// NETWORK 3 (disabled)
//   b_goto_Az_done: ********************************Zero Velocity***************************************
// fb_start_goto_az1(CLK := b_goto_Az_done); // R_TRIG
// b_start_goto_az R= fb_start_goto_az1.Q;
// b_moving R= fb_start_goto_az1.Q;

// NETWORK 4 (disabled)
//   b_scc_goto: the command of goto a fixed position for all axises
// fb_blink_move_az(ENABLE := b_moving, TIMELOW := t#1000ms, TIMEHIGH := t#200ms); // BLINK
// b_scc_goto := fb_blink_move_az.OUT;

// NETWORK 5 (disabled)
//   b_remote_on: in the remote mode
//   b_local_on: in the local mode
//   b_scc_goto: the command of goto a fixed position for all axises
//   v_elevation: Virtual axis "v_elevation" with axis number 8
// fb_goto_El(
//     Execute := (b_remote_on OR b_local_on) AND b_scc_goto,
//     Position := r_goto_el,
//     Velocity := 650,
//     Acceleration := 20,
//     Deceleration := 20,
//     Axis := v_elevation,
//     Active => b_active_el); // MC_MoveAbsolute
// b_goto_El_done := fb_goto_El.Done;

// NETWORK 6
//   b_remote_on: in the remote mode
//   b_local_on: in the local mode
//   b_start_goto_az_tcp: the command of goto a fixed position for all axises
//   v_FeedIndexer: Virtual axis "v_polarization" with axis number 9
fb_goto_FI(
    Execute := (b_remote_on OR b_local_on) AND b_start_goto_az_tcp,
    Distance := r_goto_FI,
    Velocity := vel_move_FI,
    Acceleration := 0.017,
    Deceleration := 0.017,
    Axis := v_FeedIndexer,
    Active => b_active_FI); // MC_MoveRelative
b_goto_FI_done := fb_goto_FI.Done;

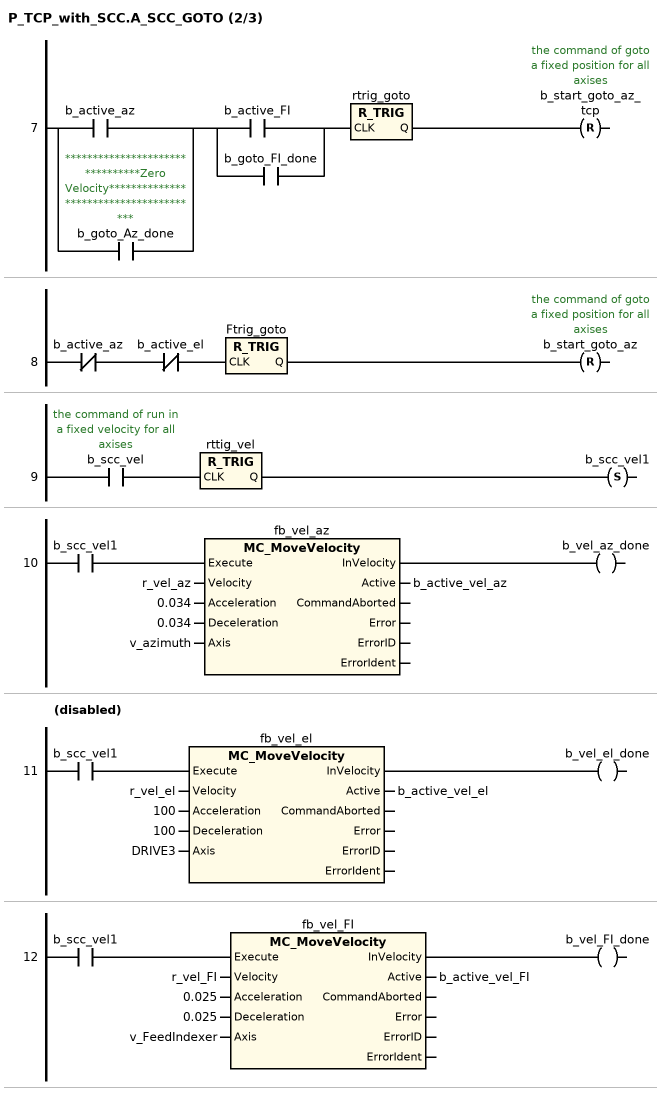
// NETWORK 7
//   b_goto_Az_done: ********************************Zero Velocity***************************************
//   b_start_goto_az_tcp: the command of goto a fixed position for all axises
rtrig_goto(CLK := (b_active_az OR b_goto_Az_done) AND (b_active_FI OR b_goto_FI_done)); // R_TRIG
b_start_goto_az_tcp R= rtrig_goto.Q;

// NETWORK 8
//   b_start_goto_az: the command of goto a fixed position for all axises
Ftrig_goto(CLK := NOT b_active_az AND NOT b_active_el); // R_TRIG
b_start_goto_az R= Ftrig_goto.Q;

// NETWORK 9
//   b_scc_vel: the command of run in a fixed velocity for all axises
rttig_vel(CLK := b_scc_vel); // R_TRIG
b_scc_vel1 S= rttig_vel.Q;

// NETWORK 10
//   r_vel_az: ************vel*************
//   v_azimuth: Virtual axis "v_azimuth" with axis number 7
fb_vel_az(
    Execute := b_scc_vel1,
    Velocity := r_vel_az,
    Acceleration := 0.034,
    Deceleration := 0.034,
    Axis := v_azimuth,
    Active => b_active_vel_az); // MC_MoveVelocity
b_vel_az_done := fb_vel_az.InVelocity;

// NETWORK 11 (disabled)
//   DRIVE3: Virtual axis "v_elevation" with axis number 8
// fb_vel_el(
//     Execute := b_scc_vel1,
//     Velocity := r_vel_el,
//     Acceleration := 100,
//     Deceleration := 100,
//     Axis := DRIVE3,
//     Active => b_active_vel_el); // MC_MoveVelocity
// b_vel_el_done := fb_vel_el.InVelocity;

// NETWORK 12
//   v_FeedIndexer: Virtual axis "v_polarization" with axis number 9
fb_vel_FI(
    Execute := b_scc_vel1,
    Velocity := r_vel_FI,
    Acceleration := 0.025,
    Deceleration := 0.025,
    Axis := v_FeedIndexer,
    Active => b_active_vel_FI); // MC_MoveVelocity
b_vel_FI_done := fb_vel_FI.InVelocity;

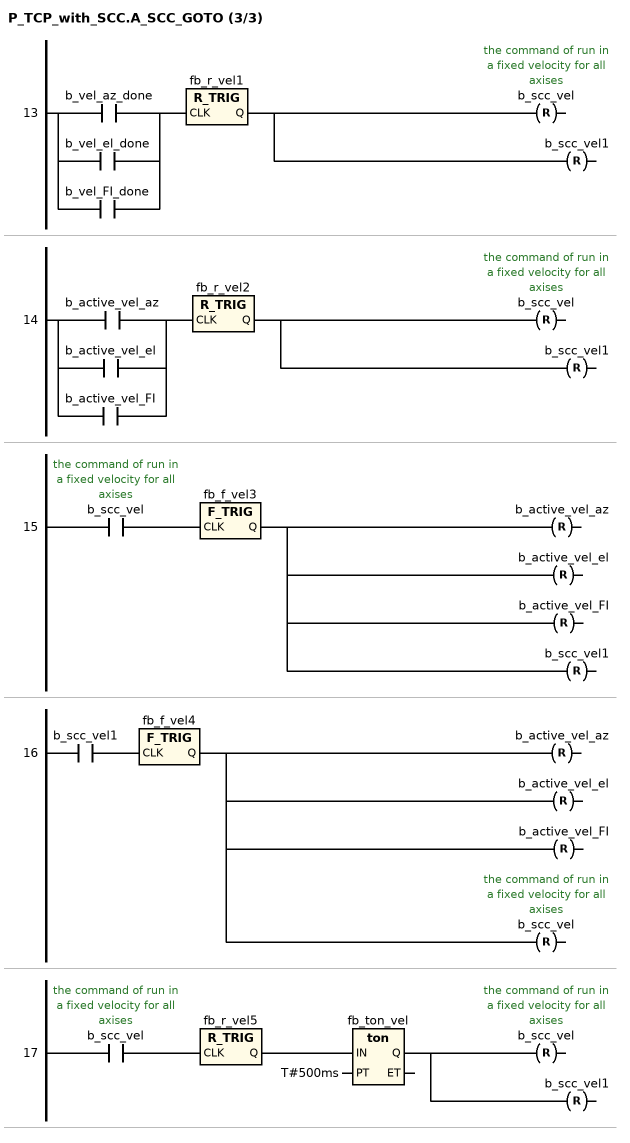
// NETWORK 13
//   b_scc_vel: the command of run in a fixed velocity for all axises
fb_r_vel1(CLK := b_vel_az_done OR b_vel_el_done OR b_vel_FI_done); // R_TRIG
b_scc_vel R= fb_r_vel1.Q;
b_scc_vel1 R= fb_r_vel1.Q;

// NETWORK 14
//   b_scc_vel: the command of run in a fixed velocity for all axises
fb_r_vel2(CLK := b_active_vel_az OR b_active_vel_el OR b_active_vel_FI); // R_TRIG
b_scc_vel R= fb_r_vel2.Q;
b_scc_vel1 R= fb_r_vel2.Q;

// NETWORK 15
//   b_scc_vel: the command of run in a fixed velocity for all axises
fb_f_vel3(CLK := b_scc_vel); // F_TRIG
b_active_vel_az R= fb_f_vel3.Q;
b_active_vel_el R= fb_f_vel3.Q;
b_active_vel_FI R= fb_f_vel3.Q;
b_scc_vel1 R= fb_f_vel3.Q;

// NETWORK 16
//   b_scc_vel: the command of run in a fixed velocity for all axises
fb_f_vel4(CLK := b_scc_vel1); // F_TRIG
b_active_vel_az R= fb_f_vel4.Q;
b_active_vel_el R= fb_f_vel4.Q;
b_active_vel_FI R= fb_f_vel4.Q;
b_scc_vel R= fb_f_vel4.Q;

// NETWORK 17
//   b_scc_vel: the command of run in a fixed velocity for all axises
fb_r_vel5(CLK := b_scc_vel); // R_TRIG
fb_ton_vel(IN := fb_r_vel5.Q, PT := T#500ms); // ton
b_scc_vel R= fb_ton_vel.Q;
b_scc_vel1 R= fb_ton_vel.Q;
END_ACTION

ACTION A_SCC_POWER:
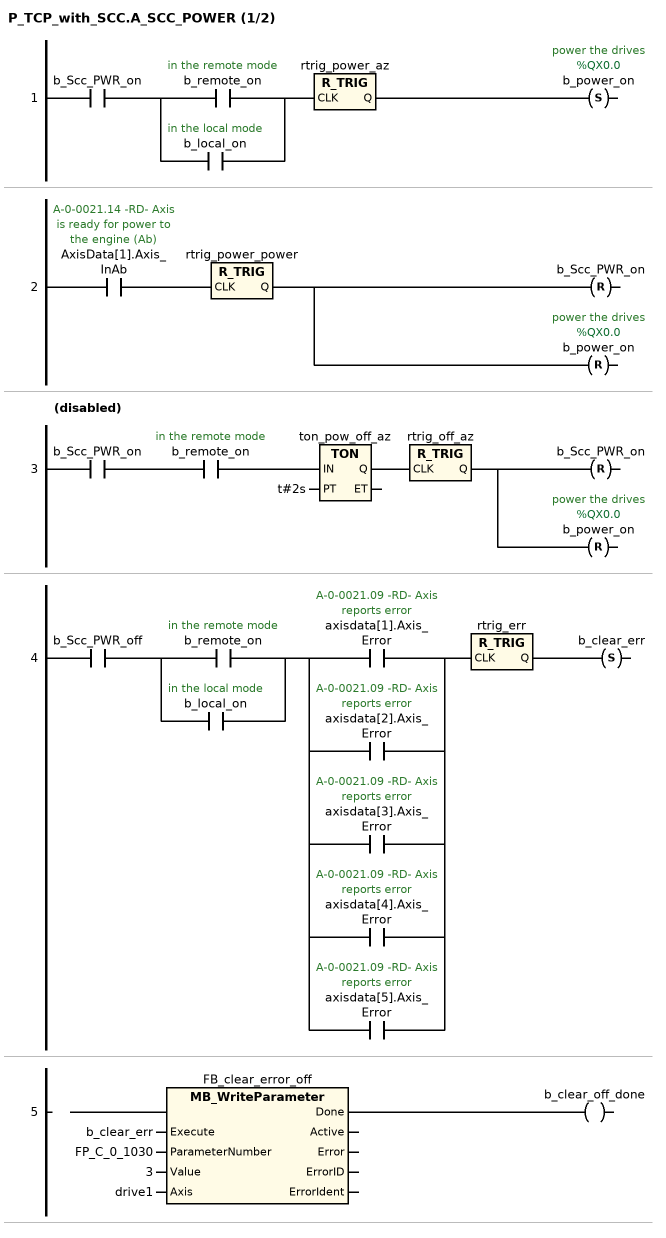
// NETWORK 1
//   b_remote_on: in the remote mode
//   b_local_on: in the local mode
//   b_power_on: power the drives | AT %QX0.0
rtrig_power_az(CLK := b_Scc_PWR_on AND (b_remote_on OR b_local_on)); // R_TRIG
b_power_on S= rtrig_power_az.Q;

// NETWORK 2
//   AxisData[1].Axis_InAb: A-0-0021.14 -RD- Axis is ready for power to the engine (Ab)
//   b_power_on: power the drives | AT %QX0.0
rtrig_power_power(CLK := AxisData[1].Axis_InAb); // R_TRIG
b_Scc_PWR_on R= rtrig_power_power.Q;
b_power_on R= rtrig_power_power.Q;

// NETWORK 3 (disabled)
//   ton_pow_off_az: <<<<<<<<<<<<<<<<<<<<<<<<<<<<<<<<<<<<<<<<<<<<<<<<<<<power>>>>>>>>>>>>>>>>>>>>>>>>>>>>>>>>>>>>
//   b_remote_on: in the remote mode
//   b_power_on: power the drives | AT %QX0.0
// ton_pow_off_az(IN := b_Scc_PWR_on AND b_remote_on, PT := t#2s); // TON
// rtrig_off_az(CLK := ton_pow_off_az.Q); // R_TRIG
// b_Scc_PWR_on R= rtrig_off_az.Q;
// b_power_on R= rtrig_off_az.Q;

// NETWORK 4
//   b_remote_on: in the remote mode
//   b_local_on: in the local mode
//   axisdata[1].Axis_Error: A-0-0021.09 -RD- Axis reports error
//   axisdata[2].Axis_Error: A-0-0021.09 -RD- Axis reports error
//   axisdata[3].Axis_Error: A-0-0021.09 -RD- Axis reports error
//   axisdata[4].Axis_Error: A-0-0021.09 -RD- Axis reports error
//   axisdata[5].Axis_Error: A-0-0021.09 -RD- Axis reports error
rtrig_err(CLK := b_Scc_PWR_off AND (b_remote_on OR b_local_on) AND (axisdata[1].Axis_Error OR axisdata[2].Axis_Error OR axisdata[3].Axis_Error OR axisdata[4].Axis_Error OR axisdata[5].Axis_Error)); // R_TRIG
b_clear_err S= rtrig_err.Q;

// NETWORK 5
//   FP_C_0_1030: Command: Clear all control errors
//   drive1: Real axis "Drive1" with axis number 1
FB_clear_error_off(Execute := b_clear_err, ParameterNumber := FP_C_0_1030, Value := 3, Axis := drive1); // MB_WriteParameter
b_clear_off_done := FB_clear_error_off.Done;

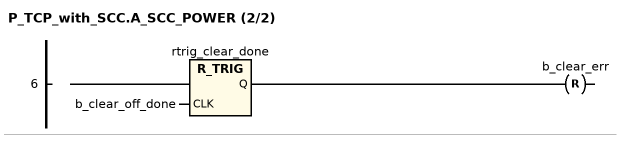
// NETWORK 6
rtrig_clear_done(CLK := b_clear_off_done); // R_TRIG
b_clear_err R= rtrig_clear_done.Q;
END_ACTION

ACTION A_SCC_STOP:
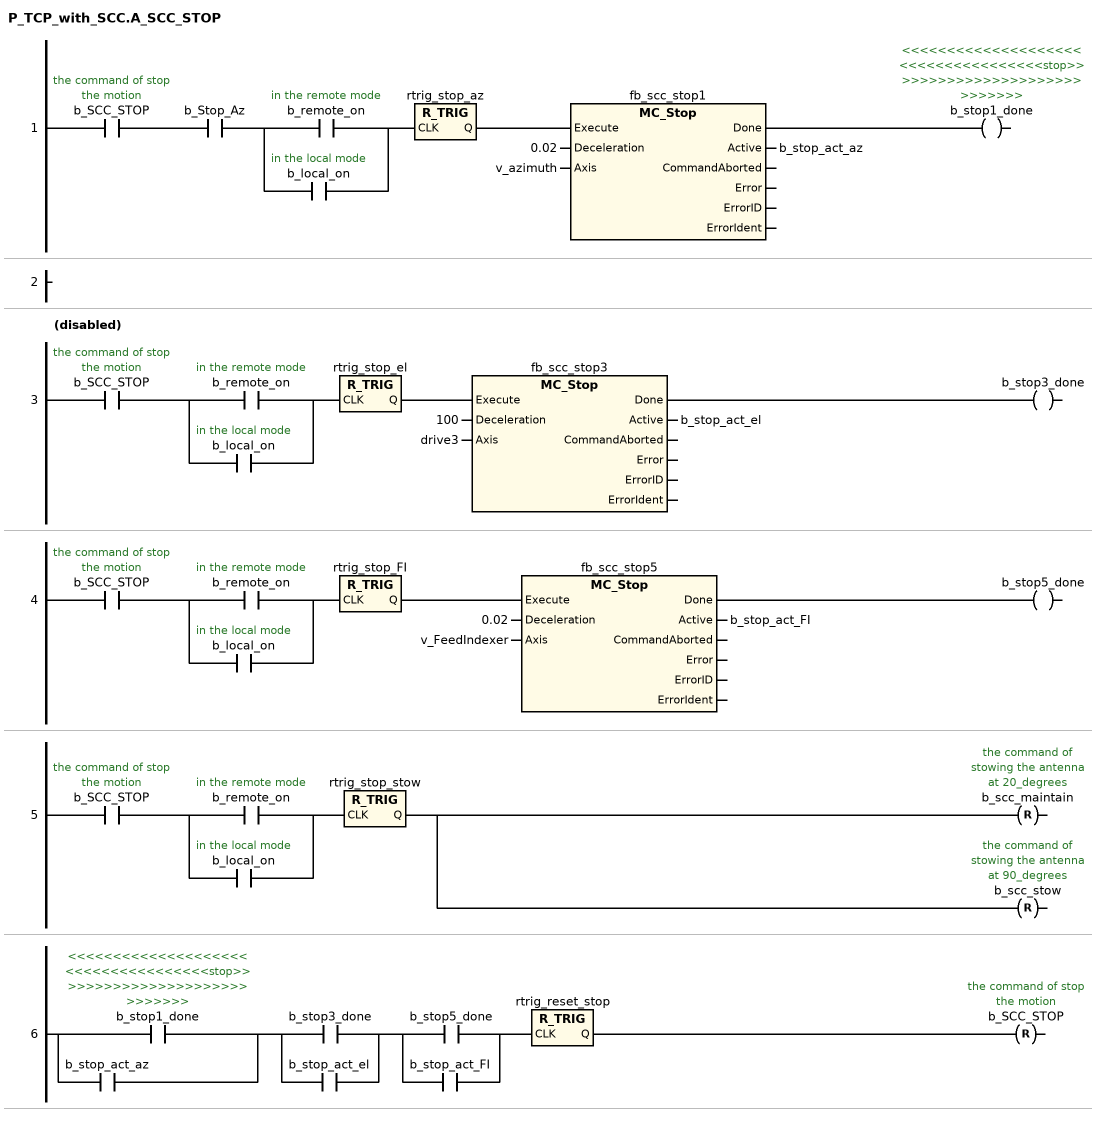
// NETWORK 1
//   b_SCC_STOP: the command of stop the motion
//   b_remote_on: in the remote mode
//   b_local_on: in the local mode
//   v_azimuth: Virtual axis "v_azimuth" with axis number 7
//   b_stop1_done: <<<<<<<<<<<<<<<<<<<<<<<<<<<<<<<<<<<<stop>>>>>>>>>>>>>>>>>>>>>>>>>>>>>
rtrig_stop_az(CLK := b_SCC_STOP AND b_Stop_Az AND (b_remote_on OR b_local_on)); // R_TRIG
fb_scc_stop1(Execute := rtrig_stop_az.Q, Deceleration := 0.02, Axis := v_azimuth, Active => b_stop_act_az); // MC_Stop
b_stop1_done := fb_scc_stop1.Done;

// NETWORK 2

// NETWORK 3 (disabled)
//   b_SCC_STOP: the command of stop the motion
//   b_remote_on: in the remote mode
//   b_local_on: in the local mode
//   drive3: Virtual axis "v_elevation" with axis number 8
// rtrig_stop_el(CLK := b_SCC_STOP AND (b_remote_on OR b_local_on)); // R_TRIG
// fb_scc_stop3(Execute := rtrig_stop_el.Q, Deceleration := 100, Axis := drive3, Active => b_stop_act_el); // MC_Stop
// b_stop3_done := fb_scc_stop3.Done;

// NETWORK 4
//   b_SCC_STOP: the command of stop the motion
//   b_remote_on: in the remote mode
//   b_local_on: in the local mode
//   v_FeedIndexer: Virtual axis "v_polarization" with axis number 9
rtrig_stop_FI(CLK := b_SCC_STOP AND (b_remote_on OR b_local_on)); // R_TRIG
fb_scc_stop5(
    Execute := rtrig_stop_FI.Q,
    Deceleration := 0.02,
    Axis := v_FeedIndexer,
    Active => b_stop_act_FI); // MC_Stop
b_stop5_done := fb_scc_stop5.Done;

// NETWORK 5
//   b_SCC_STOP: the command of stop the motion
//   b_remote_on: in the remote mode
//   b_local_on: in the local mode
//   b_scc_maintain: the command of stowing the antenna at 20_degrees
//   b_scc_stow: the command of stowing the antenna at 90_degrees
rtrig_stop_stow(CLK := b_SCC_STOP AND (b_remote_on OR b_local_on)); // R_TRIG
b_scc_maintain R= rtrig_stop_stow.Q;
b_scc_stow R= rtrig_stop_stow.Q;

// NETWORK 6
//   b_stop1_done: <<<<<<<<<<<<<<<<<<<<<<<<<<<<<<<<<<<<stop>>>>>>>>>>>>>>>>>>>>>>>>>>>>>
//   b_SCC_STOP: the command of stop the motion
rtrig_reset_stop(CLK := (b_stop1_done OR b_stop_act_az) AND (b_stop3_done OR b_stop_act_el) AND (b_stop5_done OR b_stop_act_FI)); // R_TRIG
b_SCC_STOP R= rtrig_reset_stop.Q;
END_ACTION

ACTION A_SEND:
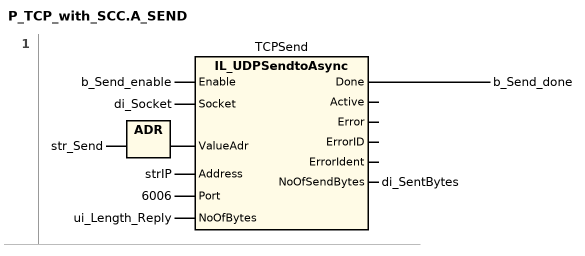
// NETWORK 1
TCPSend(
    Enable := b_Send_enable,
    Socket := di_Socket,
    ValueAdr := ADR(str_Send),
    Address := strIP,
    Port := 6006,
    NoOfBytes := ui_Length_Reply,
    NoOfSendBytes => di_SentBytes); // IL_UDPSendtoAsync
b_Send_done := TCPSend.Done;
END_ACTION

END_PROGRAM

// IndraMotionMlc1/Application/POUs/TCP/Message/FB_add_vector
(* the function block is programmed for adding points to trajectory stack.
The input variables is type of string,and the output vaiable is the reply for TCP*)
FUNCTION_BLOCK FB_add_vector
VAR_INPUT
	str_MJD:STRING;
	str_Azimuth:STRING;
	str_Elevation:STRING;
	str_FeedIndexer:STRING;
END_VAR
VAR_OUTPUT
	key:STRING;
END_VAR
VAR
(*(<<<<<<<<<<the transition variables>>>>>>>>>>>>>*)
	lreal_MJD: LREAL;
	real_azimuth: LREAL;
	real_elevation: LREAL;
	real_FeedIndexer: LREAL;
	tempAz:LREAL;
	tempEl:LREAL;
	temp_sin_Ao_C4:LREAL;
	temp_cos_Ao_C4:LREAL;
	temp_tanEo: LREAL;
	temp_sinE0:LREAL;
	temp_cosE0:LREAL;
	temp1:LREAL;
	temp2:LREAL;
	temp_R_sin_Ao_C4:LREAL;
	temp_R_cos_Ao_C4:LREAL;
	temp_R_tanEo:LREAL;
	temp_R_cosE0:LREAL;
	temp_R_sinE0:LREAL;
	temp1_exp:LREAL;
	temp2_exp:LREAL;
	new_Az:LREAL;
	new_El:LREAL;
	k:DINT;
	deltaAZ:LREAL:=0.0;
	deltaEL:LREAL:=0.0;
	aaaa:LREAL;
	bbbb:LREAL;
	test_1: LREAL;
END_VAR

(*lreal_MJD:=STRING_TO_LREAL(str_MJD)-0.000000076;*)(*set the ahead time for 6.6ms,so that the following error will be 0*)
// Assuming that for SKAO lreal_MJD will contain the TAIoffset. 
lreal_MJD:=STRING_TO_LREAL(str_MJD);(*after gunner change P41 into 100ms,so the aheed time must be added by 50ms.(56.5ms)*)

real_azimuth:=STRING_TO_LREAL(str_Azimuth);
real_Elevation:=STRING_TO_LREAL(str_Elevation);
real_FeedIndexer:=STRING_TO_REAL(str_FeedIndexer);
deltaAZ:=0.0;
deltaEL:=0.0;
	tempAz:=real_azimuth;
    tempEl:=real_Elevation;
(* This pointing model is not used for SKAO 
  		FOR k:=1 TO 3 BY 1 DO
        temp_sin_Ao_C4:=SIN(deg2rad(tempAz-C4));
        temp_cos_Ao_C4:=COS(deg2rad(tempAz-C4));
        temp_tanEo:=TAN(deg2rad(tempEl));
        temp_cosE0:=COS(deg2rad(tempEl));
        temp_sinE0:=SIN(deg2rad(tempEl));
        temp1:=tempAz-(C1+C3*temp_sin_Ao_C4*temp_tanEo+C5*temp_tanEo+C6/temp_cosE0);
        temp2:=tempEl-(C2+C3*temp_cos_Ao_C4+C7*temp_cosE0);
        temp_R_sin_Ao_C4:=SIN(deg2rad(temp1-C4));
        temp_R_cos_Ao_C4:=COS(deg2rad(temp1-C4));
        temp_R_tanEo:=TAN(deg2rad(temp2));
        temp_R_cosE0:=COS(deg2rad(temp2));
        temp_R_sinE0:=SIN(deg2rad(temp2));
        temp1_exp:=temp1+C1+C3*temp_R_sin_Ao_C4*temp_R_tanEo+C5*temp_R_tanEo+C6/temp_R_cosE0;
        temp2_exp:=temp2+C2+C3*temp_R_cos_Ao_C4+C7*temp_R_cosE0;
        deltaAz:=real_azimuth-temp1_exp;
        deltaEl:=real_Elevation-temp2_exp;
        tempAz:=tempAz+deltaAz;
        tempEl:=tempEl+deltaEl;
    END_FOR;
	*)
	new_Az:=temp1;
//	new_El:=Encoder_to_motor(temp2);
	new_El:=temp2;
	aaaa:=new_Az-real_azimuth;
	bbbb:=new_El-real_Elevation;
(*<<<<<<<<<<<<<<<<<<<<<<<<<<<<<<<judgement according to ICD document>>>>>>>>>>>>>>>>>>>>>>>>>>>>>>>*)

test_1:=lreal_MJD-lr_TAIoffset_current;
IF (lreal_MJD-lr_TAIoffset_current)>0.001 THEN	
IF real_azimuth>=-270 AND real_azimuth<=270 AND real_elevation>=15 AND real_elevation<=90 AND real_FeedIndexer>=0 AND real_FeedIndexer<=180 THEN
	IF lreal_MJD> (track_table[i_End].TAIoffset) THEN
		IF i_num_stack_left<i_total THEN
			IF track_table[i_end].TAIoffset<>0 THEN
				i_end:=F_I_number(i_end+1);
			END_IF;
			key:='OK';
			track_table[i_End].TAIoffset:=lreal_MJD;
			track_table[i_End].Azimuth:= new_Az;//-0.2884;
			track_table[i_End].Elevation:= real_Elevation;
			//track_table[i_End].FeedIndexer:= tempEl;
			//track_table[i_End].Elevation_ori:=temp2;
		ELSE
			key:='NAK - Stack is full';
		END_IF;
	ELSE
		key:='NAK - MJD is out of sequence';
	END_IF;
ELSE
	key:='NAK - One or more trkval coords are unreachable';
END_IF;
END_IF;

(*test_1:=lreal_MJD-lr_MJD_current;
IF (lreal_MJD-lr_MJD_current)>0.001 THEN	
IF real_azimuth>=-270 AND real_azimuth<=270 AND real_elevation>=15 AND real_elevation<=90 AND real_FeedIndexer>=0 AND real_FeedIndexer<=180 THEN
	IF lreal_MJD> (track_table[i_End].MJD) THEN
		IF i_num_stack_left<i_total THEN
			IF track_table[i_end].MJD<>0 THEN
				i_end:=F_I_number(i_end+1);
			END_IF;
			key:='OK';
			track_table[i_End].MJD:=lreal_MJD;
			track_table[i_End].Azimuth:= new_Az;//-0.2884;
			track_table[i_End].Elevation:= real_Elevation;
			track_table[i_End].FeedIndexer:= tempEl;
			track_table[i_End].Elevation_ori:=temp2;
		ELSE
			key:='NAK - Stack is full';
		END_IF;
	ELSE
		key:='NAK - MJD is out of sequence';
	END_IF;
ELSE
	key:='NAK - One or more trkval coords are unreachable';
END_IF;
END_IF; *)

END_FUNCTION_BLOCK

// IndraMotionMlc1/Application/AxisInterface/_Readme
PROGRAM _Readme
VAR
END_VAR

;
(*  English                              | Deutsch
Please do not change the programs and    | Bitte die Programme und Funktionsbausteine
function blocks in this folder. Updates  | in diesem Ordner nicht veraendern. Updates des
of the AxisInterface example project     | AxisInterface Besipielprojektes werden eine
will include an EXPORT-File with the     | EXPORT-Datei mit dem Inhalt dieses Ordners enthalten.
content of this folder.                  |
If you want to adapt the POUs, copy and  | Bei Anpassungen an den POEs bitte kopieren und 
rename it to avoid overwriting           | umbenennen, um ein Ueberschreiben zu vermeiden  *)

END_PROGRAM

// IndraMotionMlc1/Application/POUs/Useless/POU_1MS_Az_freq
PROGRAM POU_1MS_Az_freq
VAR
	r_cycle_count: INT;
	R_TRIG_count: R_TRIG;
	R_TRIG_count_1: R_TRIG;
	r_cycle_count_1: INT;
	MB_AxisDistanceAccumulator_1: MB_AxisDistanceAccumulator;
	bDisenable: BOOL;
	
	btestStart: BOOL;
	rdistance: REAL;
	
	CTU_1: CTU;
	bReset: BOOL;
	bSTOPPPP: BOOL;
	iTestint: REAL;
	rdistancediff: REAL;
	rdiffdistance: REAL;
	rOldDistance: REAL;
	bHometest: BOOL;
	MB_WriteRealParameter_1: MB_WriteRealParameter;
	rIniEncoderPos: REAL;

	R_TRIG_IniPos: R_TRIG;
	bStartRecord: BOOL;
	R_TRIG_condition: R_TRIG;
	teetet: BOOL;
	TON_1: TON;
	rAxis3ActVel: REAL;
	rSetAxis3Vel: REAL;
	
	R_TRIG_VEL: R_TRIG;
	test_motor_degree: LREAL;
	test_encoder: LREAL;
	
	postion_vel_array:ARRAY[1..201] OF LREAL;
	MJD_vel_array:ARRAY[1..201] OF LREAL;
	pos_vel_avg_array:ARRAY[1..181] OF LREAL;
	position_vel_i:INT:=0;
	position_vel_avg_i:INT:=0;
	position_vel_i_before:INT;
	r_temp1_pos:LREAL;
	r_temp1_mjd:LREAL;
	i_temp:INT;
	sum_vel:REAL;


	i_avg_1:INT:=0;
	i_avg_2:INT:=0;
	i_avg_3:INT:=0;
	temp_vel_avg_array:ARRAY[1..21] OF LREAL;
	sum_temp_vel:REAL;
	test1_temp:REAL;
	r_new_cmd_pos:REAL;
	r_new_cmd_pos_motor:REAL;
	r_new_cmd_pos_motor_relative:REAL;
	R_TRIG_pos_done:R_TRIG;
	R_TRIG_pos_done_2:R_TRIG;
	R_TRIG_pos_done_3:R_TRIG;
	R_TRIG_pos_done_4:R_TRIG;
	R_TRIG_pos_done_5:R_TRIG;
	R_TRIG_pos_done_6:R_TRIG;
	R_TRIG_pos_done_7:R_TRIG;
	R_TRIG_pos_done_8:R_TRIG;
	R_TRIG_pos_done_9:R_TRIG;
	R_TRIG_pos_done_10:R_TRIG;
	ton_pos2:TON;
	
	i_closeloop_max:INT:=10;
	i_time:INT:=0;
	r_difference:REAL;
	test_POWER_EL: BOOL;
	vel_blink:Util.BLINK;
	rSPEED1: REAL;
	ton_start_adjust_vel:TON;
	r_trig_start_adjust_vel: R_TRIG;
	r_vel_el_1:REAL;
	
	vel_freq:REAL;
	T_period:REAL:=2;
	temp_t:REAL:=0.0;
	start_to_freq:BOOL;
	temp_i:INT:=0;
	
	b_test_freq_resp: BOOL;
	b_in_normal_mode: BOOL := TRUE;
	b_test_pos_freq: BOOL;
	
	Frequency_vel:REAL:=0.5;
	test_vel_az1: REAL;
	A_sin:REAL;
END_VAR



	position_vel_i:= position_vel_i+1;
	IF position_vel_i>200 THEN
		position_vel_i:=1;
	END_IF
	postion_vel_array[position_vel_i]:=r_pos_el;
	MJD_vel_array[position_vel_i]:=lr_MJD_current;
	
	position_vel_i_before:=position_vel_i-100;
	IF position_vel_i_before<0 THEN
		position_vel_i_before:=position_vel_i_before+200;
	END_IF
	IF position_vel_i_before=0 THEN
		position_vel_i_before:=200;
	END_IF
		
	r_temp1_pos:=postion_vel_array[position_vel_i]-postion_vel_array[position_vel_i_before];
	r_temp1_mjd:=(MJD_vel_array[position_vel_i]-MJD_vel_array[position_vel_i_before])*86400;
	IF r_temp1_mjd= 0 THEN
		r_temp1_mjd :=1;
	END_IF
	position_vel_avg_i:=position_vel_avg_i+1;
	pos_vel_avg_array[position_vel_avg_i]:=r_temp1_pos/r_temp1_mjd;
	
	IF position_vel_avg_i = 180 THEN
		position_vel_avg_i:=0;
	END_IF
	
		sum_vel:=0;
	FOR i_temp :=1 TO 180 BY 1 DO
		sum_vel:=sum_vel+pos_vel_avg_array[i_temp];
	END_FOR
		r_vel_EL_temp:=sum_vel/180;
		
	i_avg_1:=i_avg_1+1;
	
	IF i_avg_1 =200 THEN
		i_avg_1:=0;
		i_avg_2:=i_avg_2+1;
		temp_vel_avg_array[i_avg_2]:=r_vel_EL_temp;
		IF i_avg_2>20 THEN
			i_avg_2:=0;
		END_IF		
	END_IF
	
		sum_temp_vel:=0;
	FOR i_avg_3 :=1 TO 20 BY 1 DO
		sum_temp_vel:=sum_temp_vel+temp_vel_avg_array[i_avg_3];
	END_FOR
		r_vel_EL:=sum_temp_vel/20;
	

		
	
	
//	r_vel_EL:=r_temp1_pos/r_temp1_mjd;
//	r_vel_EL:=(postion_vel_array[position_vel_i]-postion_vel_array[position_vel_i_before])/(MJD_vel_array[position_vel_i]-MJD_vel_array[position_vel_i_before])/86400;
	
	
	
	test_motor_degree:=Encoder_to_motor(test_encoder);
 
	//俯仰电机实时位置	
	r_pos_motor3:=axisdata[3].rActualPosition_i;	
	
	//俯仰电机位置累计
    rPosdiff:=RIL_Utilities.IL_GetModuloType04((axisdata[3].rActualPosition_i-roldposition),210000);
	//rPosdiff:=r_pos_motor3-roldposition;
	roldposition:=r_pos_motor3;
	r_length:=r_length+rPosdiff;
	
	CTU_1(CU:=axisdata[3].rActualPosition_i>180 , RESET:= bReset, PV:=10000 , Q=> , CV=> );
	CTU_1.CV;
	//测量Delta杆长值
	r_length_count := r_length/360/16.8*25;	
	
	//理论杆长
	Inir_Length:=SQRT(2984.1*2984.1+3150.6*3150.6-2*2984.1*3150.6*COS(r_pos_el*3.1415926/180));
	
	MB_AxisDistanceAccumulator_1(
	Enable:= bDisenable, 
	TotalDistance:= 1000000, 
	InOperation=> , 
	Error=> , 
	ErrorID=> , 
	ErrorIdent=> , 
	DistanceReached=> , 
	AccumulatedDistance=> r_length_Distance, 
	Axis:= Drive3);
/////////////**********上电设置编码器位置************////////////	
	R_TRIG_condition(CLK:=NOT TechBase.ImcStatus.Diag.Error 
							AND NOT arAxisStatus_gb[3].Admin.MODE_AH 
								AND ML_Base.AxisData[3].Axis_Inbb
									AND NOT bStartRecord, Q=> );
	IF  R_TRIG_condition.Q OR teetet  THEN 
		bHometest:=TRUE;
	END_IF
		MB_WriteRealParameter_1(
		Execute:= bHometest, 
		Done=> , 
		Active=> , 
		Error=> , 
		ErrorID=> , 
		ErrorIdent=> , 
		ParameterNumber:= ML_Base.FP_S_0_0052, 
		Value:= r_pos_motor3_Ini, 
		Axis:=Drive3 );	
	arAxisCtrl_gb[3].Admin.SetAbsRef:=MB_WriteRealParameter_1.Done;
		TON_1(IN:= MB_WriteRealParameter_1.Done, PT:=T#3S , Q=> , ET=> );
	//	R_TRIG_IniPos(CLK:= TON_1.Q, Q=> );
		IF TON_1.Q THEN 
			bStartRecord:=TRUE;
			bHometest:=FALSE;
		END_IF
		IF bStartRecord THEN
			r_pos_motor3_Ini:=axisdata[3].rActualPosition_i;
		END_IF
/////////////////**************************//////////////////////////	
 (*SIN_Curve  	
   iTestint:=iTestint+0.05;
   rdistance:=3600*SIN(iTestint*3.1415926/180);
   rdiffdistance:=rdistance-rOldDistance;
   rOldDistance:=rdistance;
   *) 
   
R_TRIG_VEL(CLK:=P_TCP_with_SCC.b_scc_vel1 , Q=> );	
IF R_TRIG_VEL.Q THEN 
	b_scc_vel1_temp:=TRUE;
END_IF

R_TRIG_pos_done(CLK:=arAxisStatus_gb[Drive3.AxisNo].Admin.CmdDone , Q=> );	
IF R_TRIG_pos_done.Q THEN 
	b_first_pos_done:=TRUE;
END_IF

R_TRIG_pos_done_2(CLK:=(arAxisStatus_gb[Drive3.AxisNo].Admin.CmdDone AND i_adjust_count=1) , Q=> );	
IF R_TRIG_pos_done_2.Q THEN 
	b_second_pos_done:=TRUE;
END_IF

R_TRIG_pos_done_3(CLK:=(arAxisStatus_gb[Drive3.AxisNo].Admin.CmdDone AND i_adjust_count=2) , Q=> );	
IF R_TRIG_pos_done_3.Q THEN 
	b_3rd_pos_done:=TRUE;
END_IF

R_TRIG_pos_done_4(CLK:=(arAxisStatus_gb[Drive3.AxisNo].Admin.CmdDone AND i_adjust_count=3) , Q=> );	
IF R_TRIG_pos_done_4.Q THEN 
	b_4th_pos_done:=TRUE;
END_IF

R_TRIG_pos_done_5(CLK:=(arAxisStatus_gb[Drive3.AxisNo].Admin.CmdDone AND i_adjust_count=4) , Q=> );	
IF R_TRIG_pos_done_5.Q THEN 
	b_5th_pos_done:=TRUE;
END_IF

R_TRIG_pos_done_6(CLK:=(arAxisStatus_gb[Drive3.AxisNo].Admin.CmdDone AND i_adjust_count=5) , Q=> );	
IF R_TRIG_pos_done_6.Q THEN 
	b_6th_pos_done:=TRUE;
END_IF

R_TRIG_pos_done_7(CLK:=(arAxisStatus_gb[Drive3.AxisNo].Admin.CmdDone AND i_adjust_count=6) , Q=> );	
IF R_TRIG_pos_done_7.Q THEN 
	b_7th_pos_done:=TRUE;
END_IF

R_TRIG_pos_done_8(CLK:=(arAxisStatus_gb[Drive3.AxisNo].Admin.CmdDone AND i_adjust_count=7) , Q=> );	
IF R_TRIG_pos_done_8.Q THEN 
	b_8th_pos_done:=TRUE;
END_IF

R_TRIG_pos_done_9(CLK:=(arAxisStatus_gb[Drive3.AxisNo].Admin.CmdDone AND i_adjust_count=8) , Q=> );	
IF R_TRIG_pos_done_9.Q THEN 
	b_9th_pos_done:=TRUE;
END_IF

R_TRIG_pos_done_10(CLK:=(arAxisStatus_gb[Drive3.AxisNo].Admin.CmdDone AND i_adjust_count=9) , Q=> );	
IF R_TRIG_pos_done_10.Q THEN 
	b_10th_pos_done:=TRUE;
END_IF

ton_pos2(IN:=b_second_pos_done,PT:=T#10S);
IF ton_pos2.Q THEN
adjust_delay:=TRUE;
END_IF

i_time:=i_time+1;
IF i_time>100 THEN
	i_time:=0;
END_IF

//IF i_time = 50 THEN
	IF TRUE THEN
	r_difference:=ABS(r_goto_el_I-r_pos_el);

IF b_in_positionMode  AND b_first_pos_done AND i_adjust_count=0 AND r_difference>0.0005 THEN

	r_new_cmd_pos:=2*r_goto_el_I-r_pos_el;
	r_new_cmd_pos_motor:=Encoder_to_motor(r_new_cmd_pos);
	r_new_cmd_pos_motor_relative:=Encoder_to_motor(r_goto_el_I)-Encoder_to_motor(ML_Base.AxisData[11].rActualPosition_i);
	r_goto_el_abs:=r_new_cmd_pos_motor;
	r_goto_el:=r_new_cmd_pos_motor_relative;
	b_in_positionMode:=FALSE;
	b_first_pos_done:=FALSE;
	b_second_pos_done:=FALSE;
	b_3rd_pos_done:=FALSE;
	b_4th_pos_done:=FALSE;
	b_5th_pos_done:=FALSE;
	b_6th_pos_done:=FALSE;
	b_7th_pos_done:=FALSE;
	b_8th_pos_done:=FALSE;
	b_9th_pos_done:=FALSE;
	b_10th_pos_done:=FALSE;
	i_adjust_count:=1;	
END_IF

IF i_adjust_count=1  AND b_second_pos_done AND  r_difference>0.0005 THEN

	r_new_cmd_pos:=2*r_goto_el_I-r_pos_el;
	r_new_cmd_pos_motor:=Encoder_to_motor(r_new_cmd_pos);
	r_new_cmd_pos_motor_relative:=Encoder_to_motor(r_goto_el_I)-Encoder_to_motor(ML_Base.AxisData[11].rActualPosition_i);
	r_goto_el_abs:=r_new_cmd_pos_motor;
	r_goto_el:=r_new_cmd_pos_motor_relative;
	b_in_positionMode:=FALSE;
	b_first_pos_done:=FALSE;
	b_second_pos_done:=FALSE;
	b_3rd_pos_done:=FALSE;
	b_4th_pos_done:=FALSE;
	b_5th_pos_done:=FALSE;
	b_6th_pos_done:=FALSE;
	b_7th_pos_done:=FALSE;
	b_8th_pos_done:=FALSE;
	b_9th_pos_done:=FALSE;
	b_10th_pos_done:=FALSE;
	adjust_delay:=FALSE;
	i_adjust_count:=2;
END_IF

IF i_adjust_count=2  AND b_3rd_pos_done AND r_difference>0.0005  THEN

	r_new_cmd_pos:=2*r_goto_el_I-r_pos_el;
	r_new_cmd_pos_motor:=Encoder_to_motor(r_new_cmd_pos);
	r_new_cmd_pos_motor_relative:=Encoder_to_motor(r_goto_el_I)-Encoder_to_motor(ML_Base.AxisData[11].rActualPosition_i);
	r_goto_el_abs:=r_new_cmd_pos_motor;
	r_goto_el:=r_new_cmd_pos_motor_relative;
	b_in_positionMode:=FALSE;
	b_first_pos_done:=FALSE;
	b_second_pos_done:=FALSE;
	b_3rd_pos_done:=FALSE;
	b_4th_pos_done:=FALSE;
	b_5th_pos_done:=FALSE;
	b_6th_pos_done:=FALSE;
	b_7th_pos_done:=FALSE;
	b_8th_pos_done:=FALSE;
	b_9th_pos_done:=FALSE;
	b_10th_pos_done:=FALSE;
	adjust_delay:=FALSE;
	i_adjust_count:=3;
END_IF

IF i_adjust_count=3  AND b_4th_pos_done AND r_difference>0.0005  THEN

	r_new_cmd_pos:=2*r_goto_el_I-r_pos_el;
	r_new_cmd_pos_motor:=Encoder_to_motor(r_new_cmd_pos);
	r_new_cmd_pos_motor_relative:=Encoder_to_motor(r_goto_el_I)-Encoder_to_motor(ML_Base.AxisData[11].rActualPosition_i);
	r_goto_el_abs:=r_new_cmd_pos_motor;
	r_goto_el:=r_new_cmd_pos_motor_relative;
	b_in_positionMode:=FALSE;
	b_first_pos_done:=FALSE;
	b_second_pos_done:=FALSE;
	b_3rd_pos_done:=FALSE;
	b_4th_pos_done:=FALSE;
	b_5th_pos_done:=FALSE;
	b_6th_pos_done:=FALSE;
	b_7th_pos_done:=FALSE;
	b_8th_pos_done:=FALSE;
	b_9th_pos_done:=FALSE;
	b_10th_pos_done:=FALSE;
	adjust_delay:=FALSE;
	i_adjust_count:=4;
END_IF

IF i_adjust_count=4  AND b_5th_pos_done AND r_difference>0.0005  THEN

	r_new_cmd_pos:=2*r_goto_el_I-r_pos_el;
	r_new_cmd_pos_motor:=Encoder_to_motor(r_new_cmd_pos);
	r_new_cmd_pos_motor_relative:=Encoder_to_motor(r_goto_el_I)-Encoder_to_motor(ML_Base.AxisData[11].rActualPosition_i);
	r_goto_el_abs:=r_new_cmd_pos_motor;
	r_goto_el:=r_new_cmd_pos_motor_relative;
	b_in_positionMode:=FALSE;
	b_first_pos_done:=FALSE;
	b_second_pos_done:=FALSE;
	b_3rd_pos_done:=FALSE;
	b_4th_pos_done:=FALSE;
	b_5th_pos_done:=FALSE;
	b_6th_pos_done:=FALSE;
	b_7th_pos_done:=FALSE;
	b_8th_pos_done:=FALSE;
	b_9th_pos_done:=FALSE;
	b_10th_pos_done:=FALSE;
	adjust_delay:=FALSE;
	i_adjust_count:=5;
END_IF
END_IF
(*
IF i_adjust_count=5  AND b_6th_pos_done THEN
	r_new_cmd_pos:=2*r_goto_el_I-r_pos_el;
	r_new_cmd_pos_motor:=Encoder_to_motor(r_new_cmd_pos);
	r_goto_el_abs:=r_new_cmd_pos_motor;
	b_in_positionMode:=FALSE;
	b_first_pos_done:=FALSE;
	b_second_pos_done:=FALSE;
	b_3rd_pos_done:=FALSE;
	b_4th_pos_done:=FALSE;
	b_5th_pos_done:=FALSE;
	b_6th_pos_done:=FALSE;
	b_7th_pos_done:=FALSE;
	b_8th_pos_done:=FALSE;
	b_9th_pos_done:=FALSE;
	b_10th_pos_done:=FALSE;
	adjust_delay:=FALSE;
	i_adjust_count:=6;
END_IF

IF i_adjust_count=6  AND b_7th_pos_done THEN
	r_new_cmd_pos:=2*r_goto_el_I-r_pos_el;
	r_new_cmd_pos_motor:=Encoder_to_motor(r_new_cmd_pos);
	r_goto_el_abs:=r_new_cmd_pos_motor;
	b_in_positionMode:=FALSE;
	b_first_pos_done:=FALSE;
	b_second_pos_done:=FALSE;
	b_3rd_pos_done:=FALSE;
	b_4th_pos_done:=FALSE;
	b_5th_pos_done:=FALSE;
	b_6th_pos_done:=FALSE;
	b_7th_pos_done:=FALSE;
	b_8th_pos_done:=FALSE;
	b_9th_pos_done:=FALSE;
	b_10th_pos_done:=FALSE;
	adjust_delay:=FALSE;
	i_adjust_count:=7;
END_IF

IF i_adjust_count=7  AND b_8th_pos_done THEN
	r_new_cmd_pos:=2*r_goto_el_I-r_pos_el;
	r_new_cmd_pos_motor:=Encoder_to_motor(r_new_cmd_pos);
	r_goto_el_abs:=r_new_cmd_pos_motor;
	b_in_positionMode:=FALSE;
	b_first_pos_done:=FALSE;
	b_second_pos_done:=FALSE;
	b_3rd_pos_done:=FALSE;
	b_4th_pos_done:=FALSE;
	b_5th_pos_done:=FALSE;
	b_6th_pos_done:=FALSE;
	b_7th_pos_done:=FALSE;
	b_8th_pos_done:=FALSE;
	b_9th_pos_done:=FALSE;
	b_10th_pos_done:=FALSE;
	adjust_delay:=FALSE;
	i_adjust_count:=8;
END_IF

IF i_adjust_count=8  AND b_9th_pos_done THEN
	r_new_cmd_pos:=2*r_goto_el_I-r_pos_el;
	r_new_cmd_pos_motor:=Encoder_to_motor(r_new_cmd_pos);
	r_goto_el_abs:=r_new_cmd_pos_motor;
	b_in_positionMode:=FALSE;
	b_first_pos_done:=FALSE;
	b_second_pos_done:=FALSE;
	b_3rd_pos_done:=FALSE;
	b_4th_pos_done:=FALSE;
	b_5th_pos_done:=FALSE;
	b_6th_pos_done:=FALSE;
	b_7th_pos_done:=FALSE;
	b_8th_pos_done:=FALSE;
	b_9th_pos_done:=FALSE;
	b_10th_pos_done:=FALSE;
	adjust_delay:=FALSE;
	i_adjust_count:=9;
END_IF

IF i_adjust_count=9  AND b_10th_pos_done THEN
	r_new_cmd_pos:=2*r_goto_el_I-r_pos_el;
	r_new_cmd_pos_motor:=Encoder_to_motor(r_new_cmd_pos);
	r_goto_el_abs:=r_new_cmd_pos_motor;
	b_in_positionMode:=FALSE;
	b_first_pos_done:=FALSE;
	b_second_pos_done:=FALSE;
	b_3rd_pos_done:=FALSE;
	b_4th_pos_done:=FALSE;
	b_5th_pos_done:=FALSE;
	b_6th_pos_done:=FALSE;
	b_7th_pos_done:=FALSE;
	b_8th_pos_done:=FALSE;
	b_9th_pos_done:=FALSE;
	b_10th_pos_done:=FALSE;
	adjust_delay:=FALSE;
	i_adjust_count:=10;
END_IF
*)
(*	
IF  arAxisStatus_gb[Drive3.AxisNo].Admin.CmdDone AND i_closeloop_count<i_closeloop_max THEN
	r_new_cmd_pos:=2*r_goto_el_I-r_pos_el;
	r_new_cmd_pos_motor:=Encoder_to_motor(r_new_cmd_pos);
	r_goto_el_abs:=r_new_cmd_pos_motor;
	arAxisStatus_gb[Drive3.AxisNo].Admin.CmdDone:=FALSE;
	i_closeloop_count:= i_closeloop_count+1;
END_IF
	IF i_closeloop_count>i_closeloop_max THEN
		i_closeloop_count:=i_closeloop_max;
	END_IF
*)
r_trig_start_adjust_vel(CLK:= b_scc_vel); 
IF r_trig_start_adjust_vel.Q THEN
	b_start_adjust_vel_temp:=TRUE;
END_IF

ton_start_adjust_vel(IN:=b_start_adjust_vel_temp,PT:=T#10S);
IF ton_start_adjust_vel.Q THEN
	b_start_adjust_vel_temp:=FALSE;
	b_start_adjust_vel:=TRUE;
END_IF

//	r_vel_el_1:= 0.00008*ML_Base.AxisData[11].rActualPosition_i*ML_Base.AxisData[11].rActualPosition_i - 0.0141*ML_Base.AxisData[11].rActualPosition_i + 1.6168;
//r_vel_el_1 := 0.0000000002*r_pos_el_v*r_pos_el_v*r_pos_el_v*r_pos_el_v*r_pos_el_v - 0.00000003*r_pos_el_v*r_pos_el_v*r_pos_el_v*r_pos_el_v + 0.000002*r_pos_el_v*r_pos_el_v*r_pos_el_v + 0.0001*r_pos_el_v*r_pos_el_v - 0.0187*r_pos_el_v + 1.6902;
r_vel_el_1 := 0.00000000928*r_pos_el_v*r_pos_el_v*r_pos_el_v*r_pos_el_v - 0.000002553*r_pos_el_v*r_pos_el_v*r_pos_el_v + 0.0003141*r_pos_el_v*r_pos_el_v - 0.02293*r_pos_el_v + 1.7235;
  IF start_to_freq THEN
		T_period:=1/Frequency_vel;	 
 		IF temp_t<T_period THEN
			temp_t:=temp_t+0.002;
			vel_freq:=A_sin*SIN(2*3.1415926*Frequency_vel*temp_t)/2656;
		ELSE
			temp_t:=0;
			temp_i:=temp_i+1;
			Frequency_vel:=0.5+0.05*temp_i;
			IF Frequency_vel>3 THEN
				Frequency_vel:=3;
			END_IF
		END_IF
 ELSE
		temp_t:=0;
		temp_i:=0;
		Frequency_vel:=0.5;
		vel_freq:=0;	
 END_IF	
 
IF b_scc_vel1_temp OR b_test_freq_resp THEN
	
	IF b_in_normal_mode THEN 
		arAxisCtrl_gb[Drive1.AxisNo].VelMode.Velocity := test_vel_az1;
		IF r_command_vel=0 THEN
		add_vel:=0;		
		END_IF	
	ELSE
		arAxisCtrl_gb[Drive1.AxisNo].VelMode.Velocity := vel_freq;
		IF start_to_freq = FALSE THEN
			arAxisCtrl_gb[Drive1.AxisNo].VelMode.Velocity:=0;
		END_IF		
	END_IF
			
	arAxisCtrl_gb[Drive1.AxisNo].VelMode.Acceleration := 0.05;
	arAxisCtrl_gb[Drive1.AxisNo].VelMode.Deceleration := 0.05;
	arAxisCtrl_gb[Drive1.AxisNo].Admin._OpMode.en := ModeVel;
  
ELSIF b_scc_goto THEN	
(*		arAxisCtrl_gb[Drive3.AxisNo].PosMode.Distance := rdistance;
	arAxisCtrl_gb[Drive3.AxisNo].PosMode.Velocity := rSPEED;
	arAxisCtrl_gb[Drive3.AxisNo].PosMode.Acceleration := 200;
	arAxisCtrl_gb[Drive3.AxisNo].PosMode.Deceleration := 200;
	arAxisCtrl_gb[Drive3.AxisNo].Admin._OpMode.en := TechInterface.ModePosRel;
		*)

//	arAxisCtrl_gb[Drive3.AxisNo].PosMode.Position:=r_goto_el_abs;
	arAxisCtrl_gb[Drive3.AxisNo].PosMode.Distance := r_goto_el;
	arAxisCtrl_gb[Drive3.AxisNo].PosMode.Velocity := rSPEED;
	arAxisCtrl_gb[Drive3.AxisNo].PosMode.Acceleration := rACC;
	arAxisCtrl_gb[Drive3.AxisNo].PosMode.Deceleration := rDCC;
//	arAxisCtrl_gb[Drive3.AxisNo].Admin._OpMode.en := ModePosAbs;
	arAxisCtrl_gb[Drive3.AxisNo].Admin._OpMode.en := ModePosAdd;
//	axisdata[Drive3.AxisNo].Axis_InPosition;
	arAxisStatus_gb[Drive3.AxisNo].Admin.CmdDone;
			
ELSE
	arAxisCtrl_gb[Drive1.AxisNo].Admin._OpMode.en := ModeAB;
END_IF 


IF bSTOPPPP THEN
	arAxisCtrl_gb[Drive3.AxisNo].Admin._OpMode.en := ModeAB;
END_IF



////////////******天线恒定速度运行********///////////////////////\

	
rAxis3ActVel:=ML_Base.AxisData[11].rActualVelocity_i*60000;
ML_Base.AxisData[11].rActualPosition_i;
ML_Base.AxisData[11].rActualVelocity_i;


(*
R_TRIG_VEL(CLK:=P_TCP_with_SCC.b_scc_vel1 , Q=> );	
IF R_TRIG_VEL.Q THEN 
	b_scc_vel1_temp:=TRUE;
END_IF
IF b_scc_vel1_temp THEN
	arAxisCtrl_gb[Drive3.AxisNo].VelMode.Velocity := P_TCP_with_SCC.r_vel_el;
	arAxisCtrl_gb[Drive3.AxisNo].VelMode.Acceleration := 100;
	arAxisCtrl_gb[Drive3.AxisNo].VelMode.Deceleration := 100;
	arAxisCtrl_gb[Drive3.AxisNo].Admin._OpMode.en := ModeVel;
ELSE
		arAxisCtrl_gb[Drive3.AxisNo].Admin._OpMode.en := Modeab;
END_IF 
*)

END_PROGRAM

// IndraMotionMlc1/Application/POUs/Useless/POU_1MS_old_mode
PROGRAM POU_1MS_old_mode
VAR
	r_cycle_count: INT;
	R_TRIG_count: R_TRIG;
	R_TRIG_count_1: R_TRIG;
	r_cycle_count_1: INT;
	MB_AxisDistanceAccumulator_1: MB_AxisDistanceAccumulator;
	bDisenable: BOOL;
	
	btestStart: BOOL;
	rdistance: REAL;
	
	CTU_1: CTU;
	bReset: BOOL;
	bSTOPPPP: BOOL;
	iTestint: REAL;
	rdistancediff: REAL;
	rdiffdistance: REAL;
	rOldDistance: REAL;
	bHometest: BOOL;
	MB_WriteRealParameter_1: MB_WriteRealParameter;
	rIniEncoderPos: REAL;

	R_TRIG_IniPos: R_TRIG;
	bStartRecord: BOOL;
	R_TRIG_condition: R_TRIG;
	teetet: BOOL;
	TON_1: TON;
	rAxis3ActVel: REAL;
	rSetAxis3Vel: REAL;
	
	R_TRIG_VEL: R_TRIG;
	test_motor_degree: LREAL;
	test_encoder: LREAL;
	
	postion_vel_array:ARRAY[1..201] OF LREAL;
	MJD_vel_array:ARRAY[1..201] OF LREAL;
	pos_vel_avg_array:ARRAY[1..181] OF LREAL;
	position_vel_i:INT:=0;
	position_vel_avg_i:INT:=0;
	position_vel_i_before:INT;
	r_temp1_pos:LREAL;
	r_temp1_mjd:LREAL;
	i_temp:INT;
	sum_vel:REAL;


	i_avg_1:INT:=0;
	i_avg_2:INT:=0;
	i_avg_3:INT:=0;
	temp_vel_avg_array:ARRAY[1..21] OF LREAL;
	sum_temp_vel:REAL;
	test1_temp:REAL;
	r_new_cmd_pos:REAL;
	r_new_cmd_pos_motor:REAL;
	r_new_cmd_pos_motor_relative:REAL;
	R_TRIG_pos_done:R_TRIG;
	R_TRIG_pos_done_2:R_TRIG;
	R_TRIG_pos_done_3:R_TRIG;
	R_TRIG_pos_done_4:R_TRIG;
	R_TRIG_pos_done_5:R_TRIG;
	R_TRIG_pos_done_6:R_TRIG;
	R_TRIG_pos_done_7:R_TRIG;
	R_TRIG_pos_done_8:R_TRIG;
	R_TRIG_pos_done_9:R_TRIG;
	R_TRIG_pos_done_10:R_TRIG;
	ton_pos2:TON;
	
	i_closeloop_max:INT:=10;
	i_time:INT:=0;
	r_difference:REAL;
	test_POWER_EL: BOOL;
	vel_blink:Util.BLINK;
	rSPEED1: REAL;
	ton_start_adjust_vel:TON;
	r_trig_start_adjust_vel: R_TRIG;
	r_vel_el_1:REAL;
	
	vel_freq:REAL;
	T_period:REAL:=1;
	temp_t:REAL:=0.0;
	start_to_freq:BOOL;
	temp_i:INT:=0;
	
	b_test_freq_resp: BOOL;
	b_in_normal_mode: BOOL := TRUE;
	b_test_pos_freq: BOOL;
	
	Frequency_vel:REAL:=1;
	b_test_random_array: BOOL;
	start_to_random_array: BOOL;
	i_random_count:DINT:=0;
	random_gain: REAL:=1;
	i_test_count:DINT:=0;
	vel_random_array:REAL;
	vel_random_array1:REAL;
	test_1: BOOL;
	ML_WriteCyclicVelocity_0: MC_MoveVelocity;
	test_vel: LREAL;
	test_move_done: BOOL;
	R_TRIG_0: R_TRIG;
	r_motorencoder_11: REAL;
	r_motorencoder_22: REAL;
	FB_readmotorencoder11: MB_ReadRealParameter;
	FB_readmotorencoder22: MB_ReadRealParameter;
	R_TRIG_1: R_TRIG;
	temp_t1: REAL:=0.0;
	BLINK_0: BLINK;
	b_test_freq_torque: BOOL;
	r_unbalance_torque:REAL;
	
	r_freq_test_velmode_A:REAL:=100;
	
	torque_freq:REAL;
	
	b_test_az_freq_torque: BOOL;
	test_torque: REAL;
	
	r_freq_test_torquemode_A:REAL:=20;
	b_test_az_frequence:BOOL;
	b_test_el_frequence:BOOL;
	FB_read1: MB_ReadRealParameter;
	r_drive3_s80: REAL;
	FB_read2: MB_ReadRealParameter;
	r_drive3_s81: REAL;
	FB_read3: MB_ReadRealParameter;
	r_drive3_p49: REAL;
	test_2: BOOL;
END_VAR


(*****************测试谐振**************)
(*****************第一步，打开trace程序，***
（******方位 Trace_AZ_freq_res,俯仰 Trace_EL_freq_res**************)
(*****************第二步，设定扫频幅值**************)
r_freq_test_torquemode_A;
(***********第三步，选定要测试的轴，方位和俯仰不要同时选中**********)
b_test_az_frequence;
b_test_el_frequence;

(*****************第四步，在软件界面转动到测试位置，再用速度模式转动轴，***
（******方位速度为0.1度/s,俯仰为0.03度/s**************)
(*****************第五步，trace重新开始记录**************)
(*****************第六步，启动力矩扫频**************)
b_test_freq_torque;
(**********第七步，结束扫频，trace停止记录，存盘，停止力矩扫频，轴停止速度*******)
b_test_freq_torque;







IF b_test_az_frequence AND b_test_el_frequence THEN
	b_test_az_frequence:=FALSE;
	b_test_el_frequence:=FALSE;
END_IF


axisdata[3].rActualPosition_i;

	position_vel_i:= position_vel_i+1;
	IF position_vel_i>200 THEN
		position_vel_i:=1;
	END_IF
	postion_vel_array[position_vel_i]:=r_pos_el;
	MJD_vel_array[position_vel_i]:=lr_MJD_current;
	
	position_vel_i_before:=position_vel_i-100;
	IF position_vel_i_before<0 THEN
		position_vel_i_before:=position_vel_i_before+200;
	END_IF
	IF position_vel_i_before=0 THEN
		position_vel_i_before:=200;
	END_IF
		
	r_temp1_pos:=postion_vel_array[position_vel_i]-postion_vel_array[position_vel_i_before];
	r_temp1_mjd:=(MJD_vel_array[position_vel_i]-MJD_vel_array[position_vel_i_before])*86400;
	IF r_temp1_mjd= 0 THEN
		r_temp1_mjd :=1;
	END_IF
	position_vel_avg_i:=position_vel_avg_i+1;
	pos_vel_avg_array[position_vel_avg_i]:=r_temp1_pos/r_temp1_mjd;
	
	IF position_vel_avg_i = 180 THEN
		position_vel_avg_i:=0;
	END_IF
	
		sum_vel:=0;
	FOR i_temp :=1 TO 180 BY 1 DO
		sum_vel:=sum_vel+pos_vel_avg_array[i_temp];
	END_FOR
		r_vel_EL_temp:=sum_vel/180;
		
	i_avg_1:=i_avg_1+1;
	
	IF i_avg_1 =200 THEN
		i_avg_1:=0;
		i_avg_2:=i_avg_2+1;
		temp_vel_avg_array[i_avg_2]:=r_vel_EL_temp;
		IF i_avg_2>20 THEN
			i_avg_2:=0;
		END_IF		
	END_IF
	
		sum_temp_vel:=0;
	FOR i_avg_3 :=1 TO 20 BY 1 DO
		sum_temp_vel:=sum_temp_vel+temp_vel_avg_array[i_avg_3];
	END_FOR
		r_vel_EL:=sum_temp_vel/20;
	

		
	
	
//	r_vel_EL:=r_temp1_pos/r_temp1_mjd;
//	r_vel_EL:=(postion_vel_array[position_vel_i]-postion_vel_array[position_vel_i_before])/(MJD_vel_array[position_vel_i]-MJD_vel_array[position_vel_i_before])/86400;
	
	
	
	test_motor_degree:=Encoder_to_motor(test_encoder);
 
	//俯仰电机实时位置	
	r_pos_motor3:=axisdata[3].rActualPosition_i;	
	
	//俯仰电机位置累计
    rPosdiff:=RIL_Utilities.IL_GetModuloType04((axisdata[3].rActualPosition_i-roldposition),210000);
	//rPosdiff:=r_pos_motor3-roldposition;
	roldposition:=r_pos_motor3;
	r_length:=r_length+rPosdiff;
	
	CTU_1(CU:=axisdata[3].rActualPosition_i>180 , RESET:= bReset, PV:=10000 , Q=> , CV=> );
	CTU_1.CV;
	//测量Delta杆长值
	r_length_count := r_length/360/16.8*25;	
	
	//理论杆长
	Inir_Length:=SQRT(2984.1*2984.1+3150.6*3150.6-2*2984.1*3150.6*COS(r_pos_el*3.1415926/180));
	
	MB_AxisDistanceAccumulator_1(
	Enable:= bDisenable, 
	TotalDistance:= 1000000, 
	InOperation=> , 
	Error=> , 
	ErrorID=> , 
	ErrorIdent=> , 
	DistanceReached=> , 
	AccumulatedDistance=> r_length_Distance, 
	Axis:= Drive3);
/////////////**********上电设置编码器位置************////////////	
	R_TRIG_condition(CLK:=NOT TechBase.ImcStatus.Diag.Error 
							AND NOT arAxisStatus_gb[3].Admin.MODE_AH 
								AND ML_Base.AxisData[3].Axis_Inbb
									AND NOT bStartRecord, Q=> );
	IF  R_TRIG_condition.Q OR teetet  THEN 
		bHometest:=FALSE;
	END_IF
		MB_WriteRealParameter_1(
		Execute:= bHometest, 
		Done=> , 
		Active=> , 
		Error=> , 
		ErrorID=> , 
		ErrorIdent=> , 
		ParameterNumber:= ML_Base.FP_S_0_0052, 
		Value:= r_pos_motor3_Ini, 
		Axis:=Drive3 );	
	arAxisCtrl_gb[3].Admin.SetAbsRef:=MB_WriteRealParameter_1.Done;
		TON_1(IN:= MB_WriteRealParameter_1.Done, PT:=T#3S , Q=> , ET=> );
	//	R_TRIG_IniPos(CLK:= TON_1.Q, Q=> );
		IF TON_1.Q THEN 
			bStartRecord:=TRUE;
			bHometest:=FALSE;
		END_IF
		IF bStartRecord THEN
			r_pos_motor3_Ini:=axisdata[3].rActualPosition_i;
		END_IF
/////////////////**************************//////////////////////////	
 (*SIN_Curve  	
   iTestint:=iTestint+0.05;
   rdistance:=3600*SIN(iTestint*3.1415926/180);
   rdiffdistance:=rdistance-rOldDistance;
   rOldDistance:=rdistance;
   *) 
   
R_TRIG_VEL(CLK:=P_TCP_with_SCC.b_scc_vel1 , Q=> );	
IF R_TRIG_VEL.Q THEN 
	b_scc_vel1_temp:=TRUE;
END_IF

R_TRIG_pos_done(CLK:=arAxisStatus_gb[Drive3.AxisNo].Admin.CmdDone , Q=> );	
IF R_TRIG_pos_done.Q THEN 
	b_first_pos_done:=TRUE;
END_IF

R_TRIG_pos_done_2(CLK:=(arAxisStatus_gb[Drive3.AxisNo].Admin.CmdDone AND i_adjust_count=1) , Q=> );	
IF R_TRIG_pos_done_2.Q THEN 
	b_second_pos_done:=TRUE;
END_IF

R_TRIG_pos_done_3(CLK:=(arAxisStatus_gb[Drive3.AxisNo].Admin.CmdDone AND i_adjust_count=2) , Q=> );	
IF R_TRIG_pos_done_3.Q THEN 
	b_3rd_pos_done:=TRUE;
END_IF

R_TRIG_pos_done_4(CLK:=(arAxisStatus_gb[Drive3.AxisNo].Admin.CmdDone AND i_adjust_count=3) , Q=> );	
IF R_TRIG_pos_done_4.Q THEN 
	b_4th_pos_done:=TRUE;
END_IF

R_TRIG_pos_done_5(CLK:=(arAxisStatus_gb[Drive3.AxisNo].Admin.CmdDone AND i_adjust_count=4) , Q=> );	
IF R_TRIG_pos_done_5.Q THEN 
	b_5th_pos_done:=TRUE;
END_IF

R_TRIG_pos_done_6(CLK:=(arAxisStatus_gb[Drive3.AxisNo].Admin.CmdDone AND i_adjust_count=5) , Q=> );	
IF R_TRIG_pos_done_6.Q THEN 
	b_6th_pos_done:=TRUE;
END_IF

R_TRIG_pos_done_7(CLK:=(arAxisStatus_gb[Drive3.AxisNo].Admin.CmdDone AND i_adjust_count=6) , Q=> );	
IF R_TRIG_pos_done_7.Q THEN 
	b_7th_pos_done:=TRUE;
END_IF

R_TRIG_pos_done_8(CLK:=(arAxisStatus_gb[Drive3.AxisNo].Admin.CmdDone AND i_adjust_count=7) , Q=> );	
IF R_TRIG_pos_done_8.Q THEN 
	b_8th_pos_done:=TRUE;
END_IF

R_TRIG_pos_done_9(CLK:=(arAxisStatus_gb[Drive3.AxisNo].Admin.CmdDone AND i_adjust_count=8) , Q=> );	
IF R_TRIG_pos_done_9.Q THEN 
	b_9th_pos_done:=TRUE;
END_IF

R_TRIG_pos_done_10(CLK:=(arAxisStatus_gb[Drive3.AxisNo].Admin.CmdDone AND i_adjust_count=9) , Q=> );	
IF R_TRIG_pos_done_10.Q THEN 
	b_10th_pos_done:=TRUE;
END_IF

ton_pos2(IN:=b_second_pos_done,PT:=T#2S);
IF ton_pos2.Q THEN
adjust_delay:=TRUE;
END_IF

i_time:=i_time+1;
IF i_time>500 THEN
	i_time:=0;
END_IF

//IF i_time = 50 THEN
	IF TRUE AND i_time = 50 THEN
	r_difference:=ABS(r_goto_el_I-r_pos_el);

IF b_in_positionMode  AND b_first_pos_done AND i_adjust_count=0 AND r_difference>0.0005 THEN

	r_new_cmd_pos:=2*r_goto_el_I-r_pos_el;
	r_new_cmd_pos_motor:=Encoder_to_motor(r_new_cmd_pos);
	r_new_cmd_pos_motor_relative:=Encoder_to_motor(r_goto_el_I)-Encoder_to_motor(ML_Base.AxisData[11].rActualPosition_i);
	r_goto_el_abs:=r_new_cmd_pos_motor;
	r_goto_el:=r_new_cmd_pos_motor_relative;
	b_in_positionMode:=FALSE;
	b_first_pos_done:=FALSE;
	b_second_pos_done:=FALSE;
	b_3rd_pos_done:=FALSE;
	b_4th_pos_done:=FALSE;
	b_5th_pos_done:=FALSE;
	b_6th_pos_done:=FALSE;
	b_7th_pos_done:=FALSE;
	b_8th_pos_done:=FALSE;
	b_9th_pos_done:=FALSE;
	b_10th_pos_done:=FALSE;
	i_adjust_count:=1;	
END_IF

IF i_adjust_count=1  AND b_second_pos_done AND  r_difference>0.0005 THEN

	r_new_cmd_pos:=2*r_goto_el_I-r_pos_el;
	r_new_cmd_pos_motor:=Encoder_to_motor(r_new_cmd_pos);
	r_new_cmd_pos_motor_relative:=Encoder_to_motor(r_goto_el_I)-Encoder_to_motor(ML_Base.AxisData[11].rActualPosition_i);
	r_goto_el_abs:=r_new_cmd_pos_motor;
	r_goto_el:=r_new_cmd_pos_motor_relative;
	b_in_positionMode:=FALSE;
	b_first_pos_done:=FALSE;
	b_second_pos_done:=FALSE;
	b_3rd_pos_done:=FALSE;
	b_4th_pos_done:=FALSE;
	b_5th_pos_done:=FALSE;
	b_6th_pos_done:=FALSE;
	b_7th_pos_done:=FALSE;
	b_8th_pos_done:=FALSE;
	b_9th_pos_done:=FALSE;
	b_10th_pos_done:=FALSE;
	adjust_delay:=FALSE;
	i_adjust_count:=2;
END_IF

IF i_adjust_count=2  AND b_3rd_pos_done AND r_difference>0.0005  THEN

	r_new_cmd_pos:=2*r_goto_el_I-r_pos_el;
	r_new_cmd_pos_motor:=Encoder_to_motor(r_new_cmd_pos);
	r_new_cmd_pos_motor_relative:=Encoder_to_motor(r_goto_el_I)-Encoder_to_motor(ML_Base.AxisData[11].rActualPosition_i);
	r_goto_el_abs:=r_new_cmd_pos_motor;
	r_goto_el:=r_new_cmd_pos_motor_relative;
	b_in_positionMode:=FALSE;
	b_first_pos_done:=FALSE;
	b_second_pos_done:=FALSE;
	b_3rd_pos_done:=FALSE;
	b_4th_pos_done:=FALSE;
	b_5th_pos_done:=FALSE;
	b_6th_pos_done:=FALSE;
	b_7th_pos_done:=FALSE;
	b_8th_pos_done:=FALSE;
	b_9th_pos_done:=FALSE;
	b_10th_pos_done:=FALSE;
	adjust_delay:=FALSE;
	i_adjust_count:=3;
END_IF

IF i_adjust_count=3  AND b_4th_pos_done AND r_difference>0.0005  THEN

	r_new_cmd_pos:=2*r_goto_el_I-r_pos_el;
	r_new_cmd_pos_motor:=Encoder_to_motor(r_new_cmd_pos);
	r_new_cmd_pos_motor_relative:=Encoder_to_motor(r_goto_el_I)-Encoder_to_motor(ML_Base.AxisData[11].rActualPosition_i);
	r_goto_el_abs:=r_new_cmd_pos_motor;
	r_goto_el:=r_new_cmd_pos_motor_relative;
	b_in_positionMode:=FALSE;
	b_first_pos_done:=FALSE;
	b_second_pos_done:=FALSE;
	b_3rd_pos_done:=FALSE;
	b_4th_pos_done:=FALSE;
	b_5th_pos_done:=FALSE;
	b_6th_pos_done:=FALSE;
	b_7th_pos_done:=FALSE;
	b_8th_pos_done:=FALSE;
	b_9th_pos_done:=FALSE;
	b_10th_pos_done:=FALSE;
	adjust_delay:=FALSE;
	i_adjust_count:=4;
END_IF

IF i_adjust_count=4  AND b_5th_pos_done AND r_difference>0.0005  THEN

	r_new_cmd_pos:=2*r_goto_el_I-r_pos_el;
	r_new_cmd_pos_motor:=Encoder_to_motor(r_new_cmd_pos);
	r_new_cmd_pos_motor_relative:=Encoder_to_motor(r_goto_el_I)-Encoder_to_motor(ML_Base.AxisData[11].rActualPosition_i);
	r_goto_el_abs:=r_new_cmd_pos_motor;
	r_goto_el:=r_new_cmd_pos_motor_relative;
	b_in_positionMode:=FALSE;
	b_first_pos_done:=FALSE;
	b_second_pos_done:=FALSE;
	b_3rd_pos_done:=FALSE;
	b_4th_pos_done:=FALSE;
	b_5th_pos_done:=FALSE;
	b_6th_pos_done:=FALSE;
	b_7th_pos_done:=FALSE;
	b_8th_pos_done:=FALSE;
	b_9th_pos_done:=FALSE;
	b_10th_pos_done:=FALSE;
	adjust_delay:=FALSE;
	i_adjust_count:=1;
END_IF
END_IF
(*
IF i_adjust_count=5  AND b_6th_pos_done THEN
	r_new_cmd_pos:=2*r_goto_el_I-r_pos_el;
	r_new_cmd_pos_motor:=Encoder_to_motor(r_new_cmd_pos);
	r_goto_el_abs:=r_new_cmd_pos_motor;
	b_in_positionMode:=FALSE;
	b_first_pos_done:=FALSE;
	b_second_pos_done:=FALSE;
	b_3rd_pos_done:=FALSE;
	b_4th_pos_done:=FALSE;
	b_5th_pos_done:=FALSE;
	b_6th_pos_done:=FALSE;
	b_7th_pos_done:=FALSE;
	b_8th_pos_done:=FALSE;
	b_9th_pos_done:=FALSE;
	b_10th_pos_done:=FALSE;
	adjust_delay:=FALSE;
	i_adjust_count:=6;
END_IF

IF i_adjust_count=6  AND b_7th_pos_done THEN
	r_new_cmd_pos:=2*r_goto_el_I-r_pos_el;
	r_new_cmd_pos_motor:=Encoder_to_motor(r_new_cmd_pos);
	r_goto_el_abs:=r_new_cmd_pos_motor;
	b_in_positionMode:=FALSE;
	b_first_pos_done:=FALSE;
	b_second_pos_done:=FALSE;
	b_3rd_pos_done:=FALSE;
	b_4th_pos_done:=FALSE;
	b_5th_pos_done:=FALSE;
	b_6th_pos_done:=FALSE;
	b_7th_pos_done:=FALSE;
	b_8th_pos_done:=FALSE;
	b_9th_pos_done:=FALSE;
	b_10th_pos_done:=FALSE;
	adjust_delay:=FALSE;
	i_adjust_count:=7;
END_IF

IF i_adjust_count=7  AND b_8th_pos_done THEN
	r_new_cmd_pos:=2*r_goto_el_I-r_pos_el;
	r_new_cmd_pos_motor:=Encoder_to_motor(r_new_cmd_pos);
	r_goto_el_abs:=r_new_cmd_pos_motor;
	b_in_positionMode:=FALSE;
	b_first_pos_done:=FALSE;
	b_second_pos_done:=FALSE;
	b_3rd_pos_done:=FALSE;
	b_4th_pos_done:=FALSE;
	b_5th_pos_done:=FALSE;
	b_6th_pos_done:=FALSE;
	b_7th_pos_done:=FALSE;
	b_8th_pos_done:=FALSE;
	b_9th_pos_done:=FALSE;
	b_10th_pos_done:=FALSE;
	adjust_delay:=FALSE;
	i_adjust_count:=8;
END_IF

IF i_adjust_count=8  AND b_9th_pos_done THEN
	r_new_cmd_pos:=2*r_goto_el_I-r_pos_el;
	r_new_cmd_pos_motor:=Encoder_to_motor(r_new_cmd_pos);
	r_goto_el_abs:=r_new_cmd_pos_motor;
	b_in_positionMode:=FALSE;
	b_first_pos_done:=FALSE;
	b_second_pos_done:=FALSE;
	b_3rd_pos_done:=FALSE;
	b_4th_pos_done:=FALSE;
	b_5th_pos_done:=FALSE;
	b_6th_pos_done:=FALSE;
	b_7th_pos_done:=FALSE;
	b_8th_pos_done:=FALSE;
	b_9th_pos_done:=FALSE;
	b_10th_pos_done:=FALSE;
	adjust_delay:=FALSE;
	i_adjust_count:=9;
END_IF

IF i_adjust_count=9  AND b_10th_pos_done THEN
	r_new_cmd_pos:=2*r_goto_el_I-r_pos_el;
	r_new_cmd_pos_motor:=Encoder_to_motor(r_new_cmd_pos);
	r_goto_el_abs:=r_new_cmd_pos_motor;
	b_in_positionMode:=FALSE;
	b_first_pos_done:=FALSE;
	b_second_pos_done:=FALSE;
	b_3rd_pos_done:=FALSE;
	b_4th_pos_done:=FALSE;
	b_5th_pos_done:=FALSE;
	b_6th_pos_done:=FALSE;
	b_7th_pos_done:=FALSE;
	b_8th_pos_done:=FALSE;
	b_9th_pos_done:=FALSE;
	b_10th_pos_done:=FALSE;
	adjust_delay:=FALSE;
	i_adjust_count:=10;
END_IF
*)
(*	
IF  arAxisStatus_gb[Drive3.AxisNo].Admin.CmdDone AND i_closeloop_count<i_closeloop_max THEN
	r_new_cmd_pos:=2*r_goto_el_I-r_pos_el;
	r_new_cmd_pos_motor:=Encoder_to_motor(r_new_cmd_pos);
	r_goto_el_abs:=r_new_cmd_pos_motor;
	arAxisStatus_gb[Drive3.AxisNo].Admin.CmdDone:=FALSE;
	i_closeloop_count:= i_closeloop_count+1;
END_IF
	IF i_closeloop_count>i_closeloop_max THEN
		i_closeloop_count:=i_closeloop_max;
	END_IF
*)
r_trig_start_adjust_vel(CLK:= b_scc_vel); 
IF r_trig_start_adjust_vel.Q THEN
	b_start_adjust_vel_temp:=TRUE;
END_IF

ton_start_adjust_vel(IN:=b_start_adjust_vel_temp,PT:=T#10S);
IF ton_start_adjust_vel.Q THEN
	b_start_adjust_vel_temp:=FALSE;
	b_start_adjust_vel:=TRUE;
END_IF

//	r_vel_el_1:= 0.00008*ML_Base.AxisData[11].rActualPosition_i*ML_Base.AxisData[11].rActualPosition_i - 0.0141*ML_Base.AxisData[11].rActualPosition_i + 1.6168;
//r_vel_el_1 := 0.0000000002*r_pos_el_v*r_pos_el_v*r_pos_el_v*r_pos_el_v*r_pos_el_v - 0.00000003*r_pos_el_v*r_pos_el_v*r_pos_el_v*r_pos_el_v + 0.000002*r_pos_el_v*r_pos_el_v*r_pos_el_v + 0.0001*r_pos_el_v*r_pos_el_v - 0.0187*r_pos_el_v + 1.6902;
r_vel_el_1 := -(0.00000000007173*r_pos_el_v*r_pos_el_v*r_pos_el_v*r_pos_el_v + 0.00000003909*r_pos_el_v*r_pos_el_v*r_pos_el_v - 0.00001355*r_pos_el_v*r_pos_el_v + 0.001506*r_pos_el_v - 0.1344)/0.1;
 
(**********************以下为伪随机序列测试模块***********************)
 IF start_to_random_array THEN
	 i_test_count:=i_test_count+1;
	 IF i_test_count=25 THEN
		 i_test_count:=0;
	 END_IF
	 
	 IF i_test_count=1 THEN
		 test_1:=FALSE;
		 test_move_done:=FALSE;
	 END_IF
	 
	 IF i_test_count =3 THEN
	 	i_random_count:=i_random_count+1;
		 vel_random_array:=track_table[i_random_count].Azimuth*random_gain;
		test_1:=TRUE;		 
	 END_IF
	 
	
	 IF i_random_count= i_End THEN 
		i_random_count:=0; 
	 END_IF	
 ELSE
		vel_random_array:=0;
		i_random_count:=0;
 END_IF	
 
(******************伪随机序列测试模块结束*********************) 


(*******************以下为谐振测试模块************************)
 IF start_to_freq OR b_test_freq_torque THEN
		T_period:=1/Frequency_vel;	 
 		IF temp_t<(5*T_period) THEN
			temp_t:=temp_t+0.002;
//			vel_freq:=r_freq_test_velmode_A*SIN(2*3.1415926*Frequency_vel*temp_t);
			torque_freq:=r_freq_test_torquemode_A*SIN(2*3.1415926*Frequency_vel*temp_t);
		ELSE
			temp_t:=0;
			temp_i:=temp_i+1;
			Frequency_vel:=1+0.025*temp_i;
			IF Frequency_vel>3 THEN
				Frequency_vel:=3;
			END_IF
		END_IF
 ELSE
		temp_t:=0;
		temp_i:=0;
		Frequency_vel:=1;
		vel_freq:=0;
		torque_freq:=0;
 END_IF
(*************************谐振测试模块结束***********************)


 IF b_test_az_frequence THEN
	ML_Base.AxisData[1].dwUserCmdDataB_q.REAL_:=torque_freq; 
 END_IF
 
 
 
IF b_scc_vel1_temp OR b_test_freq_resp OR b_test_random_array OR b_test_freq_torque THEN
	
	IF b_in_normal_mode THEN 
		arAxisCtrl_gb[Drive3.AxisNo].VelMode.Velocity := P_TCP_with_SCC.r_vel_el/r_vel_el_1;
	//	arAxisCtrl_gb[Drive3.AxisNo].VelMode.Velocity := P_TCP_with_SCC.r_vel_el;
		IF r_command_vel=0 THEN
		add_vel:=0;		
		END_IF	
	ELSE
		arAxisCtrl_gb[Drive3.AxisNo].VelMode.Velocity := vel_freq;

		IF start_to_freq = FALSE AND start_to_random_array =FALSE THEN
			arAxisCtrl_gb[Drive3.AxisNo].VelMode.Velocity:=0;
		END_IF		
	END_IF
	
	IF b_test_freq_torque AND b_test_el_frequence THEN
		ML_Base.AxisData[3].dwUserCmdDataB_q.REAL_:=torque_freq;
	END_IF
			
	arAxisCtrl_gb[Drive3.AxisNo].VelMode.Acceleration := 200;
	arAxisCtrl_gb[Drive3.AxisNo].VelMode.Deceleration := 100;
	arAxisCtrl_gb[Drive3.AxisNo].Admin._OpMode.en := ModeVel;
	
  
ELSIF b_scc_goto THEN	
(*		arAxisCtrl_gb[Drive3.AxisNo].PosMode.Distance := rdistance;
	arAxisCtrl_gb[Drive3.AxisNo].PosMode.Velocity := rSPEED;
	arAxisCtrl_gb[Drive3.AxisNo].PosMode.Acceleration := 200;
	arAxisCtrl_gb[Drive3.AxisNo].PosMode.Deceleration := 200;
	arAxisCtrl_gb[Drive3.AxisNo].Admin._OpMode.en := TechInterface.ModePosRel;
		*)

//	arAxisCtrl_gb[Drive3.AxisNo].PosMode.Position:=r_goto_el_abs;
	arAxisCtrl_gb[Drive3.AxisNo].PosMode.Distance := r_goto_el;
	arAxisCtrl_gb[Drive3.AxisNo].PosMode.Velocity := rSPEED;
	arAxisCtrl_gb[Drive3.AxisNo].PosMode.Acceleration := rACC;
	arAxisCtrl_gb[Drive3.AxisNo].PosMode.Deceleration := rDCC;
//	arAxisCtrl_gb[Drive3.AxisNo].Admin._OpMode.en := ModePosAbs;
	arAxisCtrl_gb[Drive3.AxisNo].Admin._OpMode.en := TechInterface.ModePosRel;
//	axisdata[Drive3.AxisNo].Axis_InPosition;
	arAxisStatus_gb[Drive3.AxisNo].Admin.CmdDone;			
ELSE
	arAxisCtrl_gb[Drive3.AxisNo].Admin._OpMode.en := ModeAB;
END_IF 


IF bSTOPPPP THEN
	arAxisCtrl_gb[Drive3.AxisNo].Admin._OpMode.en := ModeAB;
END_IF



////////////******天线恒定速度运行********///////////////////////\

	
rAxis3ActVel:=ML_Base.AxisData[11].rActualVelocity_i*60000;
ML_Base.AxisData[11].rActualPosition_i;
ML_Base.AxisData[11].rActualVelocity_i;


(*
R_TRIG_VEL(CLK:=P_TCP_with_SCC.b_scc_vel1 , Q=> );	
IF R_TRIG_VEL.Q THEN 
	b_scc_vel1_temp:=TRUE;
END_IF
IF b_scc_vel1_temp THEN
	arAxisCtrl_gb[Drive3.AxisNo].VelMode.Velocity := P_TCP_with_SCC.r_vel_el;
	arAxisCtrl_gb[Drive3.AxisNo].VelMode.Acceleration := 100;
	arAxisCtrl_gb[Drive3.AxisNo].VelMode.Deceleration := 100;
	arAxisCtrl_gb[Drive3.AxisNo].Admin._OpMode.en := ModeVel;
ELSE
		arAxisCtrl_gb[Drive3.AxisNo].Admin._OpMode.en := Modeab;
END_IF 
*)


POU_1MS.P_Move();

ACTION P_Move:
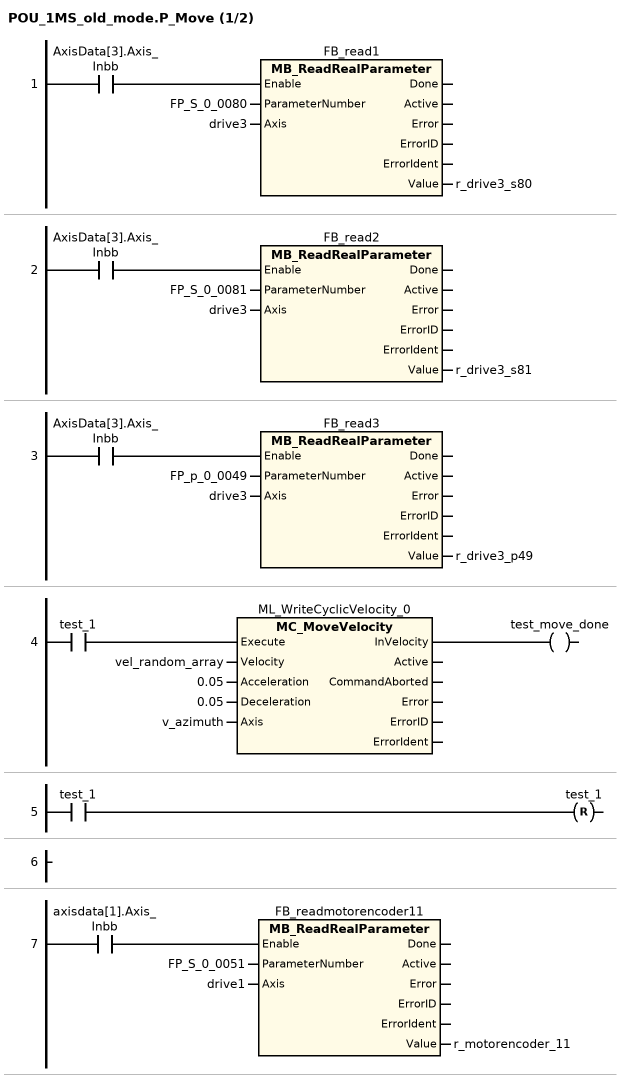
// NETWORK 1
//   FP_S_0_0080: Position feedback value 1
//   drive3: Real axis "Drive1" with axis number 1
FB_read1(
    Enable := AxisData[3].Axis_Inbb,
    ParameterNumber := FP_S_0_0080,
    Axis := drive3,
    Value => r_drive3_s80); // MB_ReadRealParameter

// NETWORK 2
//   FP_S_0_0081: Position feedback value 1
//   drive3: Real axis "Drive1" with axis number 1
FB_read2(
    Enable := AxisData[3].Axis_Inbb,
    ParameterNumber := FP_S_0_0081,
    Axis := drive3,
    Value => r_drive3_s81); // MB_ReadRealParameter

// NETWORK 3
//   FP_p_0_0049: Position feedback value 1
//   drive3: Real axis "Drive1" with axis number 1
FB_read3(
    Enable := AxisData[3].Axis_Inbb,
    ParameterNumber := FP_p_0_0049,
    Axis := drive3,
    Value => r_drive3_p49); // MB_ReadRealParameter

// NETWORK 4
ML_WriteCyclicVelocity_0(
    Execute := test_1,
    Velocity := vel_random_array,
    Acceleration := 0.05,
    Deceleration := 0.05,
    Axis := v_azimuth); // MC_MoveVelocity
test_move_done := ML_WriteCyclicVelocity_0.InVelocity;

// NETWORK 5
test_1 R= test_1;

// NETWORK 6

// NETWORK 7
//   FP_S_0_0051: Position feedback value 1
//   drive1: Real axis "Drive1" with axis number 1
FB_readmotorencoder11(
    Enable := axisdata[1].Axis_Inbb,
    ParameterNumber := FP_S_0_0051,
    Axis := drive1,
    Value => r_motorencoder_11); // MB_ReadRealParameter

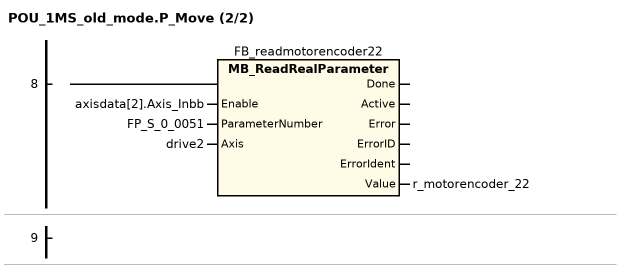
// NETWORK 8
//   axisdata[2].Axis_Inbb: A-0-0021.13 -RD- Axis is ready for power to the amplifier (bb)
//   FP_S_0_0051: Position feedback value 1
//   drive2: Real axis "Drive2" with axis number 2
FB_readmotorencoder22(
    Enable := axisdata[2].Axis_Inbb,
    ParameterNumber := FP_S_0_0051,
    Axis := drive2,
    Value => r_motorencoder_22); // MB_ReadRealParameter

// NETWORK 9
END_ACTION

END_PROGRAM

// IndraMotionMlc1/Application/POUs/Motion/POU_1MS
PROGRAM POU_1MS
VAR
	r_cycle_count: INT;
	R_TRIG_count: R_TRIG;
	R_TRIG_count_1: R_TRIG;
	r_cycle_count_1: INT;
	MB_AxisDistanceAccumulator_1: MB_AxisDistanceAccumulator;
	bDisenable: BOOL;
	
	btestStart: BOOL;
	rdistance: REAL;
	
	CTU_1: CTU;
	bReset: BOOL;
	bSTOPPPP: BOOL;
	iTestint: REAL;
	rdistancediff: REAL;
	rdiffdistance: REAL;
	rOldDistance: REAL;
	bHometest: BOOL;
	MB_WriteRealParameter_1: MB_WriteRealParameter;
	rIniEncoderPos: REAL;

	R_TRIG_IniPos: R_TRIG;
	bStartRecord: BOOL;
	R_TRIG_condition: R_TRIG;
	teetet: BOOL;
	TON_1: TON;
	rAxis3ActVel: REAL;
	rSetAxis3Vel: REAL;
	
	R_TRIG_VEL: R_TRIG;
	test_motor_degree: LREAL;
	test_encoder: LREAL;
	
	postion_vel_array:ARRAY[1..201] OF LREAL;
	MJD_vel_array:ARRAY[1..201] OF LREAL;
	pos_vel_avg_array:ARRAY[1..181] OF LREAL;
	position_vel_i:INT:=0;
	position_vel_avg_i:INT:=0;
	position_vel_i_before:INT;
	r_temp1_pos:LREAL;
	r_temp1_mjd:LREAL;
	i_temp:INT;
	sum_vel:LREAL;


	i_avg_1:INT:=0;
	i_avg_2:INT:=0;
	i_avg_3:INT:=0;
	temp_vel_avg_array:ARRAY[1..21] OF LREAL;
	sum_temp_vel:LREAL;
	test1_temp:LREAL;
	r_new_cmd_pos:LREAL;
	r_new_cmd_pos_motor:LREAL;
	r_new_cmd_pos_motor_relative:LREAL;
	R_TRIG_pos_done:R_TRIG;
	R_TRIG_pos_done_2:R_TRIG;
	R_TRIG_pos_done_3:R_TRIG;
	R_TRIG_pos_done_4:R_TRIG;
	R_TRIG_pos_done_5:R_TRIG;
	R_TRIG_pos_done_6:R_TRIG;
	R_TRIG_pos_done_7:R_TRIG;
	R_TRIG_pos_done_8:R_TRIG;
	R_TRIG_pos_done_9:R_TRIG;
	R_TRIG_pos_done_10:R_TRIG;
	ton_pos2:TON;
	
	i_closeloop_max:INT:=10;
	i_time:INT:=0;
	r_difference:LREAL;
	test_POWER_EL: BOOL;
	vel_blink:Util.BLINK;
	rSPEED1: LREAL;
	ton_start_adjust_vel:TON;
	r_trig_start_adjust_vel: R_TRIG;
	r_vel_el_1:LREAL;
	
	vel_freq:LREAL;
	T_period:LREAL:=1;
	temp_t:LREAL:=0.0;
	start_to_freq:BOOL;
	temp_i:INT:=0;
	
	b_test_freq_resp: BOOL;
	b_in_normal_mode: BOOL := TRUE;
	b_test_pos_freq: BOOL;
	
	Frequency_vel:LREAL:=0.4;
	b_test_random_array: BOOL;
	start_to_random_array: BOOL;
	i_random_count:DINT:=0;
	random_gain: LREAL:=1;
	i_test_count:DINT:=0;
	vel_random_array:LREAL;
	vel_random_array1:LREAL;
	test_1: BOOL;
	ML_WriteCyclicVelocity_0: MC_MoveVelocity;
	test_vel: LREAL;
	test_move_done: BOOL;
	R_TRIG_0: R_TRIG;
	r_motorencoder_11: LREAL;
	r_motorencoder_22: LREAL;
	FB_readmotorencoder11: MB_ReadRealParameter;
	FB_readmotorencoder22: MB_ReadRealParameter;
	R_TRIG_1: R_TRIG;
	temp_t1: LREAL:=0.0;
	BLINK_0: BLINK;
	b_test_freq_torque: BOOL;
	r_unbalance_torque:LREAL;
	
	r_freq_test_velmode_A:LREAL:=100;
	
	torque_freq:LREAL;
	
	b_test_az_freq_torque: BOOL;
	test_torque: LREAL;
	
	r_freq_test_torquemode_A:REAL:=20;
	b_test_az_frequence:BOOL;
	b_test_el_frequence:BOOL;
	FB_read1: MB_ReadRealParameter;
	r_drive3_s80: LREAL;
	FB_read2: MB_ReadRealParameter;
	r_drive3_s81: LREAL;
	FB_read3: MB_ReadRealParameter;
	r_drive3_p49: LREAL;
	test_2: BOOL;
	ML_OpenCyclicVelocityChannel_0: ML_OpenCyclicVelocityChannel;
	b_open_channel_el_vel_done: BOOL;
	
	FB_write_cycle_el_vel: ML_WriteCyclicVelocity;
	b_write_el_vel_done: BOOL;
	R_el_cycle_vel: r_trig;
	K_gear_ratio_vel:LREAL;
END_VAR


(*****************测试谐振**************)
(*****************第一步，打开trace程序，***
（******方位 Trace_AZ_freq_res,俯仰 Trace_EL_freq_res**************)
(*****************第二步，设定扫频幅值**************)
//r_freq_test_torquemode_A;
(***********第三步，选定要测试的轴，方位和俯仰不要同时选中**********)
//b_test_az_frequence;
//b_test_el_frequence;

(*****************第四步，在软件界面转动到测试位置，再用速度模式转动轴，***
（******方位速度为0.1度/s,俯仰为0.03度/s**************)
(*****************第五步，trace重新开始记录**************)
(*****************第六步，启动力矩扫频**************)
//b_test_freq_torque;
(**********第七步，结束扫频，trace停止记录，存盘，停止力矩扫频，轴停止速度*******)
//b_test_freq_torque;







IF b_test_az_frequence AND b_test_el_frequence THEN
	b_test_az_frequence:=FALSE;
	b_test_el_frequence:=FALSE;
END_IF


//axisdata[3].rActualPosition_i;

	position_vel_i:= position_vel_i+1;
	IF position_vel_i>200 THEN
		position_vel_i:=1;
	END_IF
	postion_vel_array[position_vel_i]:=r_pos_el;
	MJD_vel_array[position_vel_i]:=lr_MJD_current;
	
	position_vel_i_before:=position_vel_i-100;
	IF position_vel_i_before<0 THEN
		position_vel_i_before:=position_vel_i_before+200;
	END_IF
	IF position_vel_i_before=0 THEN
		position_vel_i_before:=200;
	END_IF
		
	r_temp1_pos:=postion_vel_array[position_vel_i]-postion_vel_array[position_vel_i_before];
	r_temp1_mjd:=(MJD_vel_array[position_vel_i]-MJD_vel_array[position_vel_i_before])*86400;
	IF r_temp1_mjd= 0 THEN
		r_temp1_mjd :=1;
	END_IF
	position_vel_avg_i:=position_vel_avg_i+1;
	pos_vel_avg_array[position_vel_avg_i]:=r_temp1_pos/r_temp1_mjd;
	
	IF position_vel_avg_i = 180 THEN
		position_vel_avg_i:=0;
	END_IF
	
		sum_vel:=0;
	FOR i_temp :=1 TO 180 BY 1 DO
		sum_vel:=sum_vel+pos_vel_avg_array[i_temp];
	END_FOR
		r_vel_EL_temp:=sum_vel/180;
		
	i_avg_1:=i_avg_1+1;
	
	IF i_avg_1 =200 THEN
		i_avg_1:=0;
		i_avg_2:=i_avg_2+1;
		temp_vel_avg_array[i_avg_2]:=r_vel_EL_temp;
		IF i_avg_2>20 THEN
			i_avg_2:=0;
		END_IF		
	END_IF
	
		sum_temp_vel:=0;
	FOR i_avg_3 :=1 TO 20 BY 1 DO
		sum_temp_vel:=sum_temp_vel+temp_vel_avg_array[i_avg_3];
	END_FOR
		r_vel_EL:=sum_temp_vel/20;
	

		
	
	
//	r_vel_EL:=r_temp1_pos/r_temp1_mjd;
//	r_vel_EL:=(postion_vel_array[position_vel_i]-postion_vel_array[position_vel_i_before])/(MJD_vel_array[position_vel_i]-MJD_vel_array[position_vel_i_before])/86400;
	
	
	
	test_motor_degree:=Encoder_to_motor(test_encoder);
 
	//俯仰电机实时位置	
	r_pos_motor3:=axisdata[3].rActualPosition_i;	
	
	//俯仰电机位置累计
    rPosdiff:=RIL_Utilities.IL_GetModuloType04((axisdata[3].rActualPosition_i-TO_REAL(roldposition)),210000);
	//rPosdiff:=r_pos_motor3-roldposition;
	roldposition:=r_pos_motor3;
	r_length:=r_length+rPosdiff;
	
	CTU_1(CU:=axisdata[3].rActualPosition_i>180 , RESET:= bReset, PV:=10000 , Q=> , CV=> );
	CTU_1.CV;
	//测量Delta杆长值
	r_length_count := r_length/360/16.8*25;	
	
	//理论杆长
	Inir_Length:=SQRT(2984.1*2984.1+3150.6*3150.6-2*2984.1*3150.6*COS(r_pos_el*3.1415926/180));
	
	MB_AxisDistanceAccumulator_1(
	Enable:= bDisenable, 
	TotalDistance:= 1000000, 
	InOperation=> , 
	Error=> , 
	ErrorID=> , 
	ErrorIdent=> , 
	DistanceReached=> , 
	AccumulatedDistance=> r_length_Distance, 
	Axis:= Drive3);
/////////////**********上电设置编码器位置************////////////	
	R_TRIG_condition(CLK:=NOT TechBase.ImcStatus.Diag.Error 
							AND NOT arAxisStatus_gb[3].Admin.MODE_AH 
								AND ML_Base.AxisData[3].Axis_Inbb
									AND NOT bStartRecord, Q=> );
	IF  R_TRIG_condition.Q OR teetet  THEN 
		bHometest:=FALSE;
	END_IF
		MB_WriteRealParameter_1(
		Execute:= bHometest, 
		Done=> , 
		Active=> , 
		Error=> , 
		ErrorID=> , 
		ErrorIdent=> , 
		ParameterNumber:= ML_Base.FP_S_0_0052, 
		Value:= r_pos_motor3_Ini, 
		Axis:=Drive3 );	
	arAxisCtrl_gb[3].Admin.SetAbsRef:=MB_WriteRealParameter_1.Done;
		TON_1(IN:= MB_WriteRealParameter_1.Done, PT:=T#3S , Q=> , ET=> );
	//	R_TRIG_IniPos(CLK:= TON_1.Q, Q=> );
		IF TON_1.Q THEN 
			bStartRecord:=TRUE;
			bHometest:=FALSE;
		END_IF
		IF bStartRecord THEN
			r_pos_motor3_Ini:=axisdata[3].rActualPosition_i;
		END_IF
/////////////////**************************//////////////////////////	
 (*SIN_Curve  	
   iTestint:=iTestint+0.05;
   rdistance:=3600*SIN(iTestint*3.1415926/180);
   rdiffdistance:=rdistance-rOldDistance;
   rOldDistance:=rdistance;
   *) 
   
R_TRIG_VEL(CLK:=P_TCP_with_SCC.b_scc_vel1 , Q=> );	
IF R_TRIG_VEL.Q THEN 
	b_scc_vel1_temp:=TRUE;
END_IF

R_TRIG_pos_done(CLK:=arAxisStatus_gb[Drive3.AxisNo].Admin.CmdDone , Q=> );	
IF R_TRIG_pos_done.Q THEN 
	b_first_pos_done:=TRUE;
END_IF

R_TRIG_pos_done_2(CLK:=(arAxisStatus_gb[Drive3.AxisNo].Admin.CmdDone AND i_adjust_count=1) , Q=> );	
IF R_TRIG_pos_done_2.Q THEN 
	b_second_pos_done:=TRUE;
END_IF

R_TRIG_pos_done_3(CLK:=(arAxisStatus_gb[Drive3.AxisNo].Admin.CmdDone AND i_adjust_count=2) , Q=> );	
IF R_TRIG_pos_done_3.Q THEN 
	b_3rd_pos_done:=TRUE;
END_IF

R_TRIG_pos_done_4(CLK:=(arAxisStatus_gb[Drive3.AxisNo].Admin.CmdDone AND i_adjust_count=3) , Q=> );	
IF R_TRIG_pos_done_4.Q THEN 
	b_4th_pos_done:=TRUE;
END_IF

R_TRIG_pos_done_5(CLK:=(arAxisStatus_gb[Drive3.AxisNo].Admin.CmdDone AND i_adjust_count=4) , Q=> );	
IF R_TRIG_pos_done_5.Q THEN 
	b_5th_pos_done:=TRUE;
END_IF

R_TRIG_pos_done_6(CLK:=(arAxisStatus_gb[Drive3.AxisNo].Admin.CmdDone AND i_adjust_count=5) , Q=> );	
IF R_TRIG_pos_done_6.Q THEN 
	b_6th_pos_done:=TRUE;
END_IF

R_TRIG_pos_done_7(CLK:=(arAxisStatus_gb[Drive3.AxisNo].Admin.CmdDone AND i_adjust_count=6) , Q=> );	
IF R_TRIG_pos_done_7.Q THEN 
	b_7th_pos_done:=TRUE;
END_IF

R_TRIG_pos_done_8(CLK:=(arAxisStatus_gb[Drive3.AxisNo].Admin.CmdDone AND i_adjust_count=7) , Q=> );	
IF R_TRIG_pos_done_8.Q THEN 
	b_8th_pos_done:=TRUE;
END_IF

R_TRIG_pos_done_9(CLK:=(arAxisStatus_gb[Drive3.AxisNo].Admin.CmdDone AND i_adjust_count=8) , Q=> );	
IF R_TRIG_pos_done_9.Q THEN 
	b_9th_pos_done:=TRUE;
END_IF

R_TRIG_pos_done_10(CLK:=(arAxisStatus_gb[Drive3.AxisNo].Admin.CmdDone AND i_adjust_count=9) , Q=> );	
IF R_TRIG_pos_done_10.Q THEN 
	b_10th_pos_done:=TRUE;
END_IF

ton_pos2(IN:=b_second_pos_done,PT:=T#2S);
IF ton_pos2.Q THEN
adjust_delay:=TRUE;
END_IF

i_time:=i_time+1;
IF i_time>500 THEN
	i_time:=0;
END_IF

//IF i_time = 50 THEN
	IF TRUE AND i_time = 50 THEN
	r_difference:=ABS(r_goto_el_I-r_pos_el);

IF b_in_positionMode  AND b_first_pos_done AND i_adjust_count=0 AND r_difference>0.0005 THEN

	r_new_cmd_pos:=2*r_goto_el_I-r_pos_el;
	r_new_cmd_pos_motor:=Encoder_to_motor(r_new_cmd_pos);
	r_new_cmd_pos_motor_relative:=Encoder_to_motor(r_goto_el_I)-Encoder_to_motor(ML_Base.AxisData[11].rActualPosition_i);
	r_goto_el_abs:=r_new_cmd_pos_motor;
	r_goto_el:=r_new_cmd_pos_motor_relative;
	b_in_positionMode:=FALSE;
	b_first_pos_done:=FALSE;
	b_second_pos_done:=FALSE;
	b_3rd_pos_done:=FALSE;
	b_4th_pos_done:=FALSE;
	b_5th_pos_done:=FALSE;
	b_6th_pos_done:=FALSE;
	b_7th_pos_done:=FALSE;
	b_8th_pos_done:=FALSE;
	b_9th_pos_done:=FALSE;
	b_10th_pos_done:=FALSE;
	i_adjust_count:=1;	
END_IF

IF i_adjust_count=1  AND b_second_pos_done AND  r_difference>0.0005 THEN

	r_new_cmd_pos:=2*r_goto_el_I-r_pos_el;
	r_new_cmd_pos_motor:=Encoder_to_motor(r_new_cmd_pos);
	r_new_cmd_pos_motor_relative:=Encoder_to_motor(r_goto_el_I)-Encoder_to_motor(ML_Base.AxisData[11].rActualPosition_i);
	r_goto_el_abs:=r_new_cmd_pos_motor;
	r_goto_el:=r_new_cmd_pos_motor_relative;
	b_in_positionMode:=FALSE;
	b_first_pos_done:=FALSE;
	b_second_pos_done:=FALSE;
	b_3rd_pos_done:=FALSE;
	b_4th_pos_done:=FALSE;
	b_5th_pos_done:=FALSE;
	b_6th_pos_done:=FALSE;
	b_7th_pos_done:=FALSE;
	b_8th_pos_done:=FALSE;
	b_9th_pos_done:=FALSE;
	b_10th_pos_done:=FALSE;
	adjust_delay:=FALSE;
	i_adjust_count:=2;
END_IF

IF i_adjust_count=2  AND b_3rd_pos_done AND r_difference>0.0005  THEN

	r_new_cmd_pos:=2*r_goto_el_I-r_pos_el;
	r_new_cmd_pos_motor:=Encoder_to_motor(r_new_cmd_pos);
	r_new_cmd_pos_motor_relative:=Encoder_to_motor(r_goto_el_I)-Encoder_to_motor(ML_Base.AxisData[11].rActualPosition_i);
	r_goto_el_abs:=r_new_cmd_pos_motor;
	r_goto_el:=r_new_cmd_pos_motor_relative;
	b_in_positionMode:=FALSE;
	b_first_pos_done:=FALSE;
	b_second_pos_done:=FALSE;
	b_3rd_pos_done:=FALSE;
	b_4th_pos_done:=FALSE;
	b_5th_pos_done:=FALSE;
	b_6th_pos_done:=FALSE;
	b_7th_pos_done:=FALSE;
	b_8th_pos_done:=FALSE;
	b_9th_pos_done:=FALSE;
	b_10th_pos_done:=FALSE;
	adjust_delay:=FALSE;
	i_adjust_count:=3;
END_IF

IF i_adjust_count=3  AND b_4th_pos_done AND r_difference>0.0005  THEN

	r_new_cmd_pos:=2*r_goto_el_I-r_pos_el;
	r_new_cmd_pos_motor:=Encoder_to_motor(r_new_cmd_pos);
	r_new_cmd_pos_motor_relative:=Encoder_to_motor(r_goto_el_I)-Encoder_to_motor(ML_Base.AxisData[11].rActualPosition_i);
	r_goto_el_abs:=r_new_cmd_pos_motor;
	r_goto_el:=r_new_cmd_pos_motor_relative;
	b_in_positionMode:=FALSE;
	b_first_pos_done:=FALSE;
	b_second_pos_done:=FALSE;
	b_3rd_pos_done:=FALSE;
	b_4th_pos_done:=FALSE;
	b_5th_pos_done:=FALSE;
	b_6th_pos_done:=FALSE;
	b_7th_pos_done:=FALSE;
	b_8th_pos_done:=FALSE;
	b_9th_pos_done:=FALSE;
	b_10th_pos_done:=FALSE;
	adjust_delay:=FALSE;
	i_adjust_count:=4;
END_IF

IF i_adjust_count=4  AND b_5th_pos_done AND r_difference>0.0005  THEN

	r_new_cmd_pos:=2*r_goto_el_I-r_pos_el;
	r_new_cmd_pos_motor:=Encoder_to_motor(r_new_cmd_pos);
	r_new_cmd_pos_motor_relative:=Encoder_to_motor(r_goto_el_I)-Encoder_to_motor(ML_Base.AxisData[11].rActualPosition_i);
	r_goto_el_abs:=r_new_cmd_pos_motor;
	r_goto_el:=r_new_cmd_pos_motor_relative;
	b_in_positionMode:=FALSE;
	b_first_pos_done:=FALSE;
	b_second_pos_done:=FALSE;
	b_3rd_pos_done:=FALSE;
	b_4th_pos_done:=FALSE;
	b_5th_pos_done:=FALSE;
	b_6th_pos_done:=FALSE;
	b_7th_pos_done:=FALSE;
	b_8th_pos_done:=FALSE;
	b_9th_pos_done:=FALSE;
	b_10th_pos_done:=FALSE;
	adjust_delay:=FALSE;
	i_adjust_count:=1;
END_IF
END_IF
(*
IF i_adjust_count=5  AND b_6th_pos_done THEN
	r_new_cmd_pos:=2*r_goto_el_I-r_pos_el;
	r_new_cmd_pos_motor:=Encoder_to_motor(r_new_cmd_pos);
	r_goto_el_abs:=r_new_cmd_pos_motor;
	b_in_positionMode:=FALSE;
	b_first_pos_done:=FALSE;
	b_second_pos_done:=FALSE;
	b_3rd_pos_done:=FALSE;
	b_4th_pos_done:=FALSE;
	b_5th_pos_done:=FALSE;
	b_6th_pos_done:=FALSE;
	b_7th_pos_done:=FALSE;
	b_8th_pos_done:=FALSE;
	b_9th_pos_done:=FALSE;
	b_10th_pos_done:=FALSE;
	adjust_delay:=FALSE;
	i_adjust_count:=6;
END_IF

IF i_adjust_count=6  AND b_7th_pos_done THEN
	r_new_cmd_pos:=2*r_goto_el_I-r_pos_el;
	r_new_cmd_pos_motor:=Encoder_to_motor(r_new_cmd_pos);
	r_goto_el_abs:=r_new_cmd_pos_motor;
	b_in_positionMode:=FALSE;
	b_first_pos_done:=FALSE;
	b_second_pos_done:=FALSE;
	b_3rd_pos_done:=FALSE;
	b_4th_pos_done:=FALSE;
	b_5th_pos_done:=FALSE;
	b_6th_pos_done:=FALSE;
	b_7th_pos_done:=FALSE;
	b_8th_pos_done:=FALSE;
	b_9th_pos_done:=FALSE;
	b_10th_pos_done:=FALSE;
	adjust_delay:=FALSE;
	i_adjust_count:=7;
END_IF

IF i_adjust_count=7  AND b_8th_pos_done THEN
	r_new_cmd_pos:=2*r_goto_el_I-r_pos_el;
	r_new_cmd_pos_motor:=Encoder_to_motor(r_new_cmd_pos);
	r_goto_el_abs:=r_new_cmd_pos_motor;
	b_in_positionMode:=FALSE;
	b_first_pos_done:=FALSE;
	b_second_pos_done:=FALSE;
	b_3rd_pos_done:=FALSE;
	b_4th_pos_done:=FALSE;
	b_5th_pos_done:=FALSE;
	b_6th_pos_done:=FALSE;
	b_7th_pos_done:=FALSE;
	b_8th_pos_done:=FALSE;
	b_9th_pos_done:=FALSE;
	b_10th_pos_done:=FALSE;
	adjust_delay:=FALSE;
	i_adjust_count:=8;
END_IF

IF i_adjust_count=8  AND b_9th_pos_done THEN
	r_new_cmd_pos:=2*r_goto_el_I-r_pos_el;
	r_new_cmd_pos_motor:=Encoder_to_motor(r_new_cmd_pos);
	r_goto_el_abs:=r_new_cmd_pos_motor;
	b_in_positionMode:=FALSE;
	b_first_pos_done:=FALSE;
	b_second_pos_done:=FALSE;
	b_3rd_pos_done:=FALSE;
	b_4th_pos_done:=FALSE;
	b_5th_pos_done:=FALSE;
	b_6th_pos_done:=FALSE;
	b_7th_pos_done:=FALSE;
	b_8th_pos_done:=FALSE;
	b_9th_pos_done:=FALSE;
	b_10th_pos_done:=FALSE;
	adjust_delay:=FALSE;
	i_adjust_count:=9;
END_IF

IF i_adjust_count=9  AND b_10th_pos_done THEN
	r_new_cmd_pos:=2*r_goto_el_I-r_pos_el;
	r_new_cmd_pos_motor:=Encoder_to_motor(r_new_cmd_pos);
	r_goto_el_abs:=r_new_cmd_pos_motor;
	b_in_positionMode:=FALSE;
	b_first_pos_done:=FALSE;
	b_second_pos_done:=FALSE;
	b_3rd_pos_done:=FALSE;
	b_4th_pos_done:=FALSE;
	b_5th_pos_done:=FALSE;
	b_6th_pos_done:=FALSE;
	b_7th_pos_done:=FALSE;
	b_8th_pos_done:=FALSE;
	b_9th_pos_done:=FALSE;
	b_10th_pos_done:=FALSE;
	adjust_delay:=FALSE;
	i_adjust_count:=10;
END_IF
*)
(*	
IF  arAxisStatus_gb[Drive3.AxisNo].Admin.CmdDone AND i_closeloop_count<i_closeloop_max THEN
	r_new_cmd_pos:=2*r_goto_el_I-r_pos_el;
	r_new_cmd_pos_motor:=Encoder_to_motor(r_new_cmd_pos);
	r_goto_el_abs:=r_new_cmd_pos_motor;
	arAxisStatus_gb[Drive3.AxisNo].Admin.CmdDone:=FALSE;
	i_closeloop_count:= i_closeloop_count+1;
END_IF
	IF i_closeloop_count>i_closeloop_max THEN
		i_closeloop_count:=i_closeloop_max;
	END_IF
*)
r_trig_start_adjust_vel(CLK:= b_scc_vel); 
IF r_trig_start_adjust_vel.Q THEN
	b_start_adjust_vel_temp:=TRUE;
END_IF

ton_start_adjust_vel(IN:=b_start_adjust_vel_temp,PT:=T#10S);
IF ton_start_adjust_vel.Q THEN
	b_start_adjust_vel_temp:=FALSE;
	b_start_adjust_vel:=TRUE;
END_IF

//	r_vel_el_1:= 0.00008*ML_Base.AxisData[11].rActualPosition_i*ML_Base.AxisData[11].rActualPosition_i - 0.0141*ML_Base.AxisData[11].rActualPosition_i + 1.6168;
//r_vel_el_1 := 0.0000000002*r_pos_el_v*r_pos_el_v*r_pos_el_v*r_pos_el_v*r_pos_el_v - 0.00000003*r_pos_el_v*r_pos_el_v*r_pos_el_v*r_pos_el_v + 0.000002*r_pos_el_v*r_pos_el_v*r_pos_el_v + 0.0001*r_pos_el_v*r_pos_el_v - 0.0187*r_pos_el_v + 1.6902;
r_vel_el_1 := -(0.00000000007173*r_pos_el_v*r_pos_el_v*r_pos_el_v*r_pos_el_v + 0.00000003909*r_pos_el_v*r_pos_el_v*r_pos_el_v - 0.00001355*r_pos_el_v*r_pos_el_v + 0.001506*r_pos_el_v - 0.1344)/0.1;
K_gear_ratio_vel:=K_gear_ratio/2000;
(**********************以下为伪随机序列测试模块***********************)
 IF start_to_random_array THEN
	 i_test_count:=i_test_count+1;
	 IF i_test_count=25 THEN
		 i_test_count:=0;
	 END_IF
	 
	 IF i_test_count=1 THEN
		 test_1:=FALSE;
		 test_move_done:=FALSE;
	 END_IF
	 
	 IF i_test_count =3 THEN
	 	i_random_count:=i_random_count+1;
		 vel_random_array:=track_table[i_random_count].Azimuth*random_gain;
		test_1:=TRUE;		 
	 END_IF
	 
	
	 IF i_random_count= i_End THEN 
		i_random_count:=0; 
	 END_IF	
 ELSE
		vel_random_array:=0;
		i_random_count:=0;
 END_IF	
 
(******************伪随机序列测试模块结束*********************) 


(*******************以下为谐振测试模块************************)
 IF start_to_freq OR b_test_freq_torque THEN
		T_period:=1/Frequency_vel;	 
 		IF temp_t<(20*T_period) THEN
			temp_t:=temp_t+0.001;
//			vel_freq:=r_freq_test_velmode_A*SIN(2*3.1415926*Frequency_vel*temp_t);
			torque_freq:=r_freq_test_torquemode_A*SIN(2*3.1415926*Frequency_vel*temp_t);
		ELSE
			temp_t:=0;
			temp_i:=temp_i+1;
			IF b_test_az_frequence THEN	
				IF Frequency_vel<1 THEN
					Frequency_vel:=0.4+0.1*temp_i;
				ELSE
					Frequency_vel:=1+0.01*(temp_i-6);
				END_IF
			END_IF	
		
			IF b_test_el_frequence THEN	
				IF Frequency_vel<1.5 THEN
					Frequency_vel:=1+0.1*temp_i;
				ELSE
					Frequency_vel:=1.5+0.05*(temp_i-5);
				END_IF
			END_IF				
			IF Frequency_vel>3.0 THEN
				Frequency_vel:=3.0;
			END_IF
		END_IF
 ELSE
		temp_t:=0;
		temp_i:=0;
		IF b_test_az_frequence THEN
			Frequency_vel:=0.4;
		END_IF
		IF b_test_EL_frequence THEN
			Frequency_vel:=1.0;
		END_IF
		vel_freq:=0;
		torque_freq:=0;
 END_IF
(*************************谐振测试模块结束***********************)


 IF b_test_az_frequence THEN
	ML_Base.AxisData[1].dwUserCmdDataB_q.REAL_:=TO_REAL(torque_freq); 
 END_IF
 
 
 
IF b_scc_vel1_temp OR b_test_freq_resp OR b_test_random_array OR b_test_freq_torque THEN
	
	IF b_in_normal_mode THEN 
		arAxisCtrl_gb[Drive3.AxisNo].VelMode.Velocity := P_TCP_with_SCC.r_vel_el/TO_REAL(r_vel_el_1);
	//	arAxisCtrl_gb[Drive3.AxisNo].VelMode.Velocity := P_TCP_with_SCC.r_vel_el*K_gear_ratio_vel;
		IF r_command_vel=0 THEN
		add_vel:=0;		
		END_IF	
	ELSE
		arAxisCtrl_gb[Drive3.AxisNo].VelMode.Velocity := TO_REAL(vel_freq);

		IF start_to_freq = FALSE AND start_to_random_array =FALSE THEN
			arAxisCtrl_gb[Drive3.AxisNo].VelMode.Velocity:=0;
		END_IF		
	END_IF
	
	IF b_test_freq_torque AND b_test_el_frequence THEN
		ML_Base.AxisData[3].dwUserCmdDataB_q.REAL_:=TO_REAL(torque_freq);
	END_IF
			
	arAxisCtrl_gb[Drive3.AxisNo].VelMode.Acceleration := 200;
	arAxisCtrl_gb[Drive3.AxisNo].VelMode.Deceleration := 100;
	arAxisCtrl_gb[Drive3.AxisNo].Admin._OpMode.en := ModeVel;
	
  
ELSIF b_scc_goto THEN
	r_following_1:=r_following_11;
	arAxisCtrl_gb[Drive3.AxisNo].Admin._OpMode.en := ModeCyclicVelocity; 
	b_write_el_vel:=TRUE;
(*

//	arAxisCtrl_gb[Drive3.AxisNo].PosMode.Position:=r_goto_el_abs;
	arAxisCtrl_gb[Drive3.AxisNo].PosMode.Distance := r_goto_el;
	arAxisCtrl_gb[Drive3.AxisNo].PosMode.Velocity := rSPEED;
	arAxisCtrl_gb[Drive3.AxisNo].PosMode.Acceleration := rACC;
	arAxisCtrl_gb[Drive3.AxisNo].PosMode.Deceleration := rDCC;
//	arAxisCtrl_gb[Drive3.AxisNo].Admin._OpMode.en := ModePosAbs;
	arAxisCtrl_gb[Drive3.AxisNo].Admin._OpMode.en := TechInterface.ModePosRel;
//	axisdata[Drive3.AxisNo].Axis_InPosition;
	arAxisStatus_gb[Drive3.AxisNo].Admin.CmdDone;
*)

			
ELSE
	arAxisCtrl_gb[Drive3.AxisNo].Admin._OpMode.en := ModeAB;
END_IF 


IF bSTOPPPP THEN
	arAxisCtrl_gb[Drive3.AxisNo].Admin._OpMode.en := ModeAB;
END_IF



////////////******天线恒定速度运行********///////////////////////\

	
rAxis3ActVel:=ML_Base.AxisData[11].rActualVelocity_i*60000;
//ML_Base.AxisData[11].rActualPosition_i;
//ML_Base.AxisData[11].rActualVelocity_i;


(*
R_TRIG_VEL(CLK:=P_TCP_with_SCC.b_scc_vel1 , Q=> );	
IF R_TRIG_VEL.Q THEN 
	b_scc_vel1_temp:=TRUE;
END_IF
IF b_scc_vel1_temp THEN
	arAxisCtrl_gb[Drive3.AxisNo].VelMode.Velocity := P_TCP_with_SCC.r_vel_el;
	arAxisCtrl_gb[Drive3.AxisNo].VelMode.Acceleration := 100;
	arAxisCtrl_gb[Drive3.AxisNo].VelMode.Deceleration := 100;
	arAxisCtrl_gb[Drive3.AxisNo].Admin._OpMode.en := ModeVel;
ELSE
		arAxisCtrl_gb[Drive3.AxisNo].Admin._OpMode.en := Modeab;
END_IF 
*)


POU_1MS.P_Move();

ACTION P_Move:
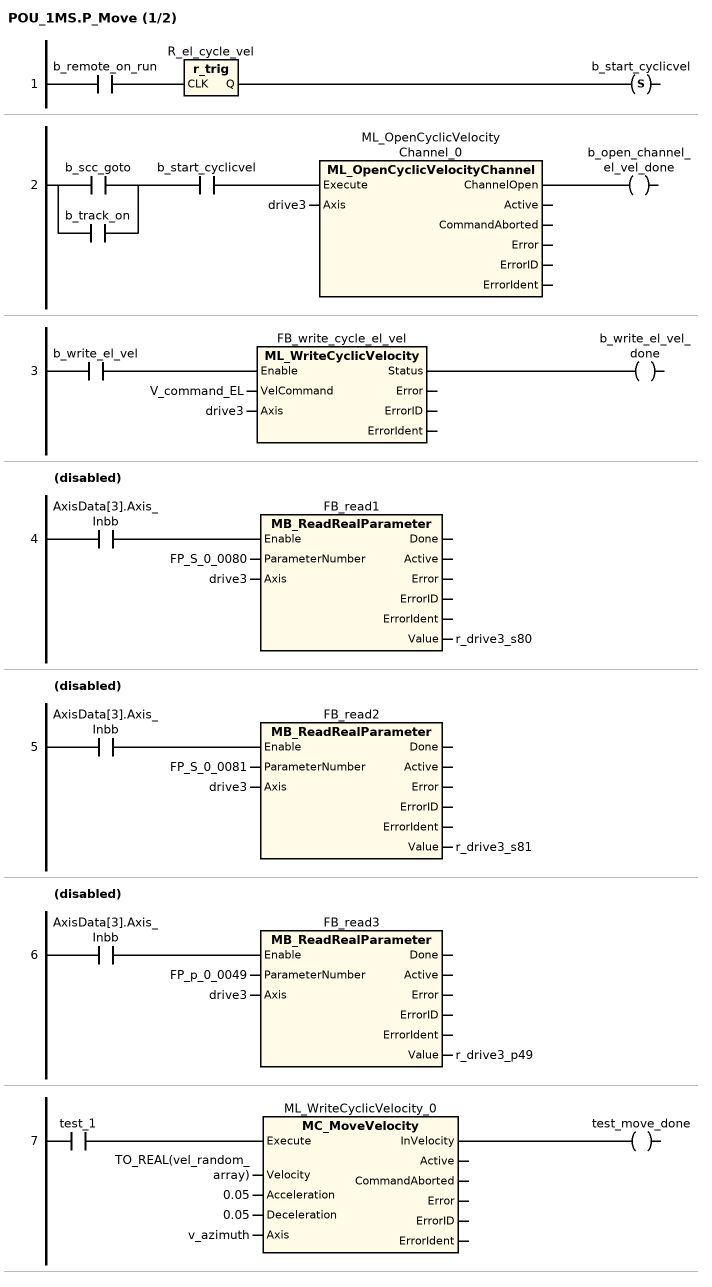
// NETWORK 1
R_el_cycle_vel(CLK := b_remote_on_run); // r_trig
b_start_cyclicvel S= R_el_cycle_vel.Q;

// NETWORK 2
ML_OpenCyclicVelocityChannel_0(Execute := (b_scc_goto OR b_track_on) AND b_start_cyclicvel, Axis := drive3); // ML_OpenCyclicVelocityChannel
b_open_channel_el_vel_done := ML_OpenCyclicVelocityChannel_0.ChannelOpen;

// NETWORK 3
FB_write_cycle_el_vel(Enable := b_write_el_vel, VelCommand := V_command_EL, Axis := drive3); // ML_WriteCyclicVelocity
b_write_el_vel_done := FB_write_cycle_el_vel.Status;

// NETWORK 4 (disabled)
//   FP_S_0_0080: Position feedback value 1
//   drive3: Real axis "Drive1" with axis number 1
// FB_read1(
//     Enable := AxisData[3].Axis_Inbb,
//     ParameterNumber := FP_S_0_0080,
//     Axis := drive3,
//     Value => r_drive3_s80); // MB_ReadRealParameter

// NETWORK 5 (disabled)
//   FP_S_0_0081: Position feedback value 1
//   drive3: Real axis "Drive1" with axis number 1
// FB_read2(
//     Enable := AxisData[3].Axis_Inbb,
//     ParameterNumber := FP_S_0_0081,
//     Axis := drive3,
//     Value => r_drive3_s81); // MB_ReadRealParameter

// NETWORK 6 (disabled)
//   FP_p_0_0049: Position feedback value 1
//   drive3: Real axis "Drive1" with axis number 1
// FB_read3(
//     Enable := AxisData[3].Axis_Inbb,
//     ParameterNumber := FP_p_0_0049,
//     Axis := drive3,
//     Value => r_drive3_p49); // MB_ReadRealParameter

// NETWORK 7
ML_WriteCyclicVelocity_0(
    Execute := test_1,
    Velocity := TO_REAL(vel_random_array),
    Acceleration := 0.05,
    Deceleration := 0.05,
    Axis := v_azimuth); // MC_MoveVelocity
test_move_done := ML_WriteCyclicVelocity_0.InVelocity;

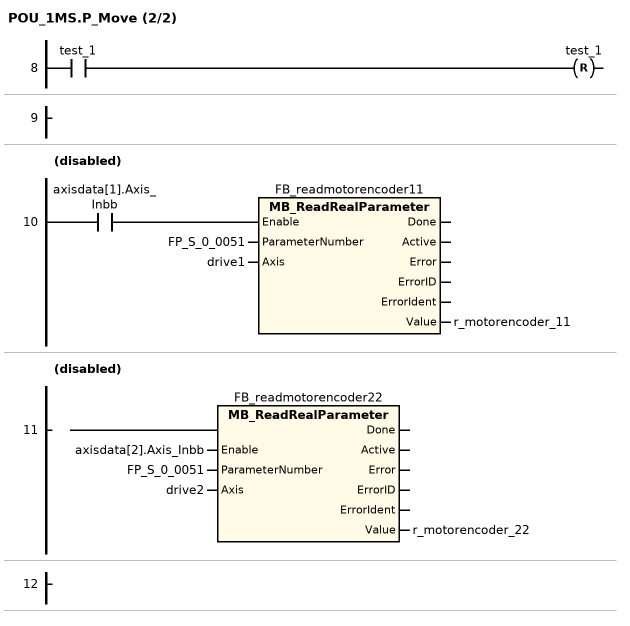
// NETWORK 8
test_1 R= test_1;

// NETWORK 9

// NETWORK 10 (disabled)
//   FP_S_0_0051: Position feedback value 1
//   drive1: Real axis "Drive1" with axis number 1
// FB_readmotorencoder11(
//     Enable := axisdata[1].Axis_Inbb,
//     ParameterNumber := FP_S_0_0051,
//     Axis := drive1,
//     Value => r_motorencoder_11); // MB_ReadRealParameter

// NETWORK 11 (disabled)
//   axisdata[2].Axis_Inbb: A-0-0021.13 -RD- Axis is ready for power to the amplifier (bb)
//   FP_S_0_0051: Position feedback value 1
//   drive2: Real axis "Drive2" with axis number 2
// FB_readmotorencoder22(
//     Enable := axisdata[2].Axis_Inbb,
//     ParameterNumber := FP_S_0_0051,
//     Axis := drive2,
//     Value => r_motorencoder_22); // MB_ReadRealParameter

// NETWORK 12
END_ACTION

END_PROGRAM

// IndraMotionMlc1/Application/POUs/TCP/Message/Encoder_to_motor_old
FUNCTION Encoder_to_motor_old : LREAL
VAR_INPUT
	encoder_input:LREAL;
END_VAR
VAR
END_VAR

(*
Encoder_to_motor:=P1*EXPT(encoder_input+40,8)+P2*EXPT(encoder_input+40,7)+P3*EXPT(encoder_input+40,6)+P4*EXPT(encoder_input+40,5)
					+P5*EXPT(encoder_input+40,4)+P6*EXPT(encoder_input+40,3)+P7*EXPT(encoder_input+40,2)
						+P8*(encoder_input+40)+P9+1000000;
*)						
Encoder_to_motor:=P1*EXPT(encoder_input,8)+P2*EXPT(encoder_input,7)+P3*EXPT(encoder_input,6)+P4*EXPT(encoder_input,5)
					+P5*EXPT(encoder_input,4)+P6*EXPT(encoder_input,3)+P7*EXPT(encoder_input,2)
						+P8*(encoder_input)+P9;

END_FUNCTION

// IndraMotionMlc1/Application/POUs/TCP/Message/FB_Caculate_position_1
FUNCTION_BLOCK FB_Caculate_position_1
VAR_INPUT
	Pos_start:LREAL;
	pos_end:LREAL;
	vel_start:LREAL;
	vel_end:LREAL;
	acc_start:LREAL;
	acc_end:LREAL;
	T_sum:LREAL;
	T_count:LREAL;			
END_VAR
VAR_OUTPUT
	cyclic_positon:LREAL;
END_VAR
VAR
	C0:LREAL;
	C1:LREAL;
	C2:LREAL;
	C3:LREAL;
	C4:LREAL;
	C5:LREAL;
	Y0:LREAL;
	Y1:LREAL;
	Y2:LREAL;
	Y3:LREAL;
	Y4:LREAL;
	Y5:LREAL;	
END_VAR

Y0:=Pos_start;
Y1:=vel_start*T_sum;
Y2:=acc_start*T_sum*T_sum/2;
Y3:=pos_end;
Y4:=vel_end*T_sum;
Y5:=acc_end*T_sum*T_sum/2;

C0:=Y0;
C1:=Y1;
C2:=Y2;
C3:=10*Y3-4*Y4+Y5-10*C0-6*C1-3*C2;
C4:=5*Y3-Y4-5*C0-4*C1-3*C2-2*C3;
C5:=Y3-C0-C1-C2-C3-C4;

cyclic_positon:=C5*EXPT(T_count,5)+C4*EXPT(T_count,4)+C3*EXPT(T_count,3)+C2*EXPT(T_count,2)+C1*T_count+C0;

END_FUNCTION_BLOCK

// IndraMotionMlc1/Application/POUs/OPCUA/OPCUA_Method/fb_Axis
(*{attribute 'opcua.mapping.type' := ''}
{attribute 'opcua.mapping.modeluri' := 'http://skao.int/DS_ICD/'}
{attribute 'opcua.mapping.publicationdate' := '12/14/2023 00:00:00'}
{attribute 'opcua.mapping.nodeid' := 'nsu=http://skao.int/DS_ICD/;i=1004'}*)

FUNCTION_BLOCK fb_Axis
VAR_INPUT 
	Status: AxisGeneralStatus_Type;
	ErrorStatus: AxisErrorStatus_Type;
	MotorOne: MotorStatus_Type;
	MotorTwo: MotorStatus_Type;
	WarningStatus: AxisWarning_Type;
END_VAR

END_FUNCTION_BLOCK

// IndraMotionMlc1/Application/POUs/OPCUA/OPCUA_Method/fb_CommandArbiter
(*{attribute 'opcua.mapping.type' := ''}
{attribute 'opcua.mapping.modeluri' := 'http://skao.int/DS_ICD/'}
{attribute 'opcua.mapping.publicationdate' := '12/14/2023 00:00:00'}
{attribute 'opcua.mapping.nodeid' := 'nsu=http://skao.int/DS_ICD/;i=1003'}*)
FUNCTION_BLOCK fb_CommandArbiter
VAR_INPUT
	Commands: fb_CommandArbiter_Commands;
	Status: CommandArbiter_Status_Type;
	    (* the authority for DSC control now 0 NoAuthority 1 LMC 2 HHP 3 EGUI*)
    Lmc_ID :UINT:=1;
	Egui_ID:UINT:=1;
	
	
END_VAR
VAR
	IL_SysTime64_0: IL_SysTime64;
	Current_time: SYS_TIME64;  
	GetTime : Bool :=1;
END_VAR

END_FUNCTION_BLOCK

// IndraMotionMlc1/Application/POUs/OPCUA/OPCUA_Method/fb_CommandArbiter_Commands
FUNCTION_BLOCK fb_CommandArbiter_Commands
VAR_INPUT
END_VAR
VAR_OUTPUT
END_VAR

VAR
	IL_SysTime64_0: IL_SysTime64;
	Current_time: SYS_TIME64;  
	GetTime : Bool :=1;

END_VAR

METHOD TakeAuth :UINT (* Take Authority *)
VAR_INPUT
	User:UINT; // 0 NoAuthority 1 LMC 2. HHP 3 EGUI 
END_VAR

VAR_OUTPUT 
	SessionID: UINT;
END_VAR
CommandArbiter.Commands.Get_Time();
IF (User >=0) AND (User <=5) THEN
	IF CommandArbiter.Status.DscCmdAuthority=HHP THEN              // If HHP is plugged in no other user can take controll
		TakeAuth:=CmdResponseType.NoCmdAuth;
		CommandArbiter.Egui_ID := 1;                            //If HHP Gets plugged in then SessionID'ds are cleared.
		CommandArbiter.Lmc_ID := 1;
		
	ELSE
		CASE User OF 
      	 1: IF CommandArbiter.Status.DscCmdAuthority=EGUI THEN      // LMC Can't take control if Egui has control
           		TakeAuth:=CmdResponseType.NoCmdAuth;   
	   	    ELSIF CommandArbiter.Lmc_ID = 1 OR CommandArbiter.Status.DscCmdAuthority= LMC THEN 
		 		CommandArbiter.Status.DscCmdAuthority:= LMC;
	     		CommandArbiter.Lmc_ID:=TO_UINT(Current_time.LowValue)+1;
				SessionID := CommandArbiter.Lmc_ID;
				CommandArbiter.Egui_ID := 1;  
				TakeAuth:=CmdResponseType.CommandDone;
		    ELSE
				//TakeAuth:=CmdResponseType.CommandFailed;
				//SessionID := 1;
		    END_IF
	   
	   	 3: IF CommandArbiter.Egui_ID = 1 OR CommandArbiter.Status.DscCmdAuthority= EGUI THEN
            	CommandArbiter.Status.DscCmdAuthority:= EGUI;           // Egui can take controll if system is in LMC control 
	        	CommandArbiter.Egui_ID:=TO_UINT(Current_time.LowValue)+1;
				SessionID := CommandArbiter.Egui_ID;
				CommandArbiter.Lmc_ID := 1;
				TakeAuth:=CmdResponseType.CommandDone;
		    ELSE 
				//TakeAuth:=CmdResponseType.CommandFailed;
				//SessionID :=2;
		    END_IF
		ELSE
	     	TakeAuth:=CmdResponseType.CommandFailed;      // Only the LMC and EGUI can Take control
         	//SessionID := 3;        			
 		END_CASE
	END_IF
ELSE 
	TakeAuth:=CmdResponseType.ParameterOutOfRange;
END_IF
CommandArbiter.Status.LastCmdResponse:= TakeAuth;
END_METHOD

METHOD ReleaseAuth :UINT
VAR_INPUT
	SessionID :UINT; 
    User : UINT;
END_VAR
CASE CommandArbiter.Status.DscCmdAuthority OF 
	 HHP: ReleaseAuth:=CmdResponseType.NoCmdAuth;
	
     LMC: IF CommandArbiter.Lmc_ID = SessionId AND User=DscCmdAuthorityType.LMC THEN 
		  	 CommandArbiter.Status.DscCmdAuthority:= NoAuthority;
	      	 CommandArbiter.Lmc_ID:=1;   
	      	 ReleaseAuth:=CmdResponseType.CommandDone;
	  	  END_IF
			
	 EGUI: IF CommandArbiter.Egui_ID = SessionID AND User=DscCmdAuthorityType.EGUI THEN
		 	  CommandArbiter.Status.DscCmdAuthority:= NoAuthority;
	      	  CommandArbiter.Egui_ID:=1;   
	      	  ReleaseAuth:=CmdResponseType.CommandDone;
	       END_IF
ELSE
     ReleaseAuth:=CmdResponseType.CommandFailed; 
END_CASE

	CommandArbiter.Status.LastCmdResponse:=ReleaseAuth;
END_METHOD

ACTION Get_Time:
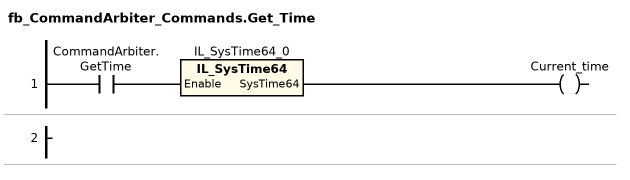
// NETWORK 1
IL_SysTime64_0(Enable := CommandArbiter.GetTime); // IL_SysTime64
Current_time := IL_SysTime64_0.SysTime64;

// NETWORK 2
END_ACTION

END_FUNCTION_BLOCK

// IndraMotionMlc1/Application/POUs/OPCUA/OPCUA_Method/fb_Management
(*{attribute 'opcua.mapping.type' := ''}
{attribute 'opcua.mapping.modeluri' := 'http://skao.int/DS_ICD/'}
{attribute 'opcua.mapping.publicationdate' := '12/14/2023 00:00:00'}
{attribute 'opcua.mapping.nodeid' := 'nsu=http://skao.int/DS_ICD/;i=1008'}*)
FUNCTION_BLOCK fb_Management
VAR_INPUT
	Commands:fb_Mngmt_Commands;
 	ErrorStatus: MngmtErrorStatus_Type;	
	NamePlate: NamePlate_Type;
	PowerStatus: PowerStatus_Type;	
	Status: MngmtStatus_Type;
	TempHumidStatus: TempHumidStatus_Type;
	WarningStatus: MngmtWarningStatus_Type;
END_VAR

END_FUNCTION_BLOCK

// IndraMotionMlc1/Application/POUs/OPCUA/OPCUA_Method/fb_Mngmt_Commands
{attribute "linkalways"}
FUNCTION_BLOCK INTERNAL fb_Mngmt_Commands
VAR_INPUT
END_VAR
VAR_OUTPUT
END_VAR
VAR
END_VAR

METHOD Activate : UINT
VAR_INPUT
	SessionID:UINT:=0;
	Axis: UINT:=3; (* 0=Az 1=El 2=FI 3=AzEl*)
	
END_VAR
VAR_OUTPUT
	
END_VAR
VAR
	
END_VAR
CASE CommandArbiter.Status.DscCmdAuthority OF                    // Check that corerct user is issueing a command
	LMC: IF SessionID= CommandArbiter.Lmc_ID THEN
			Activate:= CmdResponseType.CommandActivated;
     	 END_IF
			
	EGUI: IF SessionID= CommandArbiter.Egui_ID THEN
			Activate:= CmdResponseType.CommandActivated;
    	  END_IF		
ELSE 
     Activate:= CmdResponseType.NoCmdAuth;
     Command_Arbiter_error:=1;	
END_CASE

(*
IF Management.ErrorStatus.errGeneral = 1 THEN 
	Activate := CmdResponseType.CommandFailed;
END_IF *)

IF Activate = CmdResponseType.CommandActivated THEN
	Command_Arbiter_error:=0;
	CASE Management.Status.DscState OF 
		DSCStateType.StartUp:
		 	Activate := CmdResponseType.CommandRejected;
		DSCStateType.Standby:
		 	Activate := CmdResponseType.CommandActivated;
		DSCStateType.Locked:
		 	Activate := CmdResponseType.DishLocked;
		DSCStateType.Stowed:
		    IF Axis=2 THEN 
				Activate := CmdResponseType.CommandActivated;
			ELSE
		 	Activate :=CmdResponseType.Stowed;
			END_IF
			
		DSCStateType.Locked_Stowed:
		 	Activate := CmdResponseType.DishLocked; 
		DSCStateType.Activating :
		 	Activate := CmdResponseType.CommandActivated;
		DSCStateType.Deactivating :
		 	Activate := CmdResponseType.CommandRejected;
		DSCStateType.Standstill :
		 	Activate := CmdResponseType.CommandActivated;
		DSCStateType.Stopping :
		 	Activate := CmdResponseType.CommandActivated;
		DSCStateType.Slew :
		 	Activate := CmdResponseType.CommandActivated;
		DSCStateType.Jog :
		 	Activate := CmdResponseType.CommandActivated;
		DSCStateType.Track :
		 	Activate := CmdResponseType.CommandActivated;
	END_CASE

   IF Activate = CmdResponseType.CommandActivated THEN
	 CASE Axis OF
		AxisSelectType.Az:
			IF Management.ErrorStatus.errAzimuth=0 THEN
				b_activate_Az:=1;
				b_deactivate_Az:=0;
			ELSE 
				Activate := CmdResponseType.CommandFailed;
			END_IF
		AxisSelectType.El:
			IF Management.ErrorStatus.errElevation=0 THEN
				 b_activate_el:=1;
				 b_deactivate_El:=0;
			ELSE 
				Activate := CmdResponseType.CommandFailed;
			END_IF;
		AxisSelectType.Fi:
			IF Management.ErrorStatus.errFeedIndexer=0 THEN
				 b_activate_fi:=1;
				 b_deactivate_Fi:=0;
			ELSE 
				Activate := CmdResponseType.CommandFailed;
			END_IF;
		AxisSelectType.AzEl:
			IF Management.ErrorStatus.errAzimuth=0 AND Management.ErrorStatus.errElevation=0  THEN
				b_activate_Az:=1;
				b_deactivate_Az:=0;
				b_activate_el:=1;
				b_deactivate_el:=0;
			//	b_SCC_enable_off:=FALSE;
			//	b_SCC_enable_on:=TRUE; 
			ELSE 
				Activate := CmdResponseType.CommandFailed;
			END_IF;
		ELSE 
			//Activate := CmdResponseType.ParameterOutOfRange;
		END_CASE
   END_IF
ELSE 
	Activate := CmdResponseType.NoCmdAuth;
END_IF
CommandArbiter.Status.AxisSelect:=Axis;
CommandArbiter.Status.LastCmdResponse:=Activate;
END_METHOD

METHOD DeActivate : UINT
VAR_INPUT
	SessionID: UINT;
	Axis: UINT;
END_VAR
VAR_OUTPUT
	
END_VAR
VAR
END_VAR
CASE CommandArbiter.Status.DscCmdAuthority OF                    // Check that corerct user is issueing a command
	LMC: IF SessionID= CommandArbiter.Lmc_ID THEN
			DeActivate:= CmdResponseType.CommandActivated;
         END_IF
			
	EGUI: IF SessionID= CommandArbiter.Egui_ID THEN
			DeActivate:= CmdResponseType.CommandActivated;
          END_IF		
ELSE 
     DeActivate:= CmdResponseType.NoCmdAuth;
     Command_Arbiter_error:=1;	
END_CASE

IF DeActivate = CmdResponseType.CommandActivated THEN       // Check Dish State
	Command_Arbiter_error:=0;
	CASE Management.Status.DscState OF 
		DSCStateType.StartUp:
		 	DeActivate := CmdResponseType.CommandRejected;
		DSCStateType.Standby:
		 	DeActivate := CmdResponseType.CommandActivated;
		DSCStateType.Locked:
		 	DeActivate := CmdResponseType.DishLocked;
		DSCStateType.Stowed:
		 	DeActivate :=CmdResponseType.Stowed;
		DSCStateType.Locked_Stowed:
		 	DeActivate := CmdResponseType.DishLocked; 
		DSCStateType.Activating :
		 	DeActivate := CmdResponseType.CommandActivated;
		DSCStateType.Deactivating :
		 	DeActivate := CmdResponseType.CommandActivated;
		DSCStateType.Standstill :
		 	DeActivate := CmdResponseType.CommandActivated;
		DSCStateType.Stopping :
		 	DeActivate := CmdResponseType.CommandActivated;
		DSCStateType.Slew :
		 	DeActivate := CmdResponseType.CommandActivated;
		DSCStateType.Jog :
		 	DeActivate := CmdResponseType.CommandActivated;
		DSCStateType.Track :
		 	DeActivate := CmdResponseType.CommandActivated;
	END_CASE

   IF DeActivate = CmdResponseType.CommandActivated THEN     //Deactivate Axis
	 CASE Axis OF
		AxisSelectType.Az:
		   		b_deactivate_Az:=1;                      //Ladder logic checks for motion and stops axis before deactivating              				
				b_activate_Az:=0;             
		AxisSelectType.El:
		    	b_deactivate_El:=1;
				b_activate_el:=0;
		AxisSelectType.Fi:
		    	b_deactivate_Fi:=1;
	    		b_activate_fi:=0;
		AxisSelectType.AzEl:
		    	b_deactivate_Az:=1;
				b_deactivate_El:=1;	
				b_activate_Az:=0;
				b_activate_el:=0;
	ELSE 
		DeActivate := CmdResponseType.ParameterOutOfRange;
	END_CASE
   END_IF
ELSE 
   DeActivate:= CmdResponseType.NoCmdAuth;
END_IF
CommandArbiter.Status.LastCmdResponse:=DeActivate;
END_METHOD

METHOD Move2Band : UINT
VAR_INPUT
	SessionID : UINT;
	Band :UINT;
END_VAR
CASE CommandArbiter.Status.DscCmdAuthority OF                    // Check that correct user is issueing a command
	LMC: IF SessionID= CommandArbiter.Lmc_ID THEN
			Move2Band:= CmdResponseType.CommandActivated;
     	 END_IF
			
	EGUI: IF SessionID= CommandArbiter.Egui_ID THEN
			Move2Band:= CmdResponseType.CommandActivated;
    	  END_IF		
ELSE 
     Move2Band:= CmdResponseType.NoCmdAuth;
     Command_Arbiter_error:=1;	
END_CASE

IF Move2Band = CmdResponseType.CommandActivated THEN // Check Dish State to see if move is possible
	Command_Arbiter_error:=0;
	IF  Management.ErrorStatus.errGeneral=0 AND Management.WarningStatus.waMngmnt =0 THEN  
		CASE Management.Status.DscState OF 
			 DscStateType.Locked:        Move2Band:=CmdResponseType.DishLocked;
			 DscStateType.Locked_Stowed: Move2Band:=CmdResponseType.DishLocked;
			 DscStateType.Standstill:    Move2Band:=CmdResponseType.CommandActivated;
		     DscStateType.Standby:       Move2Band:=CmdResponseType.CommandActivated;
			 DscStateType.Stowed:	     Move2Band:=CmdResponseType.CommandActivated;
			 DscStateType.Slew:  		 Move2Band:=CmdResponseType.CommandActivated;
			 DscStateType.Track:  		 Move2Band:=CmdResponseType.CommandActivated;
			 DscStateType.Activating:	 Move2Band:=CmdResponseType.CommandActivated;
			 DscStateType.Deactivating:	 Move2Band:=CmdResponseType.CommandActivated;
			 DscStateType.Stopping:		 Move2Band:=CmdResponseType.CommandActivated;
			
		ELSE
		     Move2Band:=CmdResponseType.CommandRejected;
		     Command_Arbiter_error:=1;
		END_CASE	
   		CASE Band OF   // get band position
	 		Bandtype.Optical: r_goto_Fi := gc_r_band_optical ; 
                              FeedIndexer.Status.p_Set:= gc_r_band_optical;   
     		Bandtype.Band_1:  r_goto_Fi :=gc_r_band_1 ;
							  FeedIndexer.Status.p_Set:= gc_r_band_1;   
	 		Bandtype.Band_2:  r_goto_Fi := gc_r_band_2 ;
							  FeedIndexer.Status.p_Set:= gc_r_band_2;   
	 		Bandtype.Band_3:  r_goto_Fi := gc_r_band_3 ;
						      FeedIndexer.Status.p_Set:= gc_r_band_3;   
	 		Bandtype.Band_4:  r_goto_Fi := gc_r_band_4 ;
							  FeedIndexer.Status.p_Set:= gc_r_band_4;   
	 		Bandtype.Band_5a: r_goto_Fi := gc_r_band_5a ;
							  FeedIndexer.Status.p_Set:= gc_r_band_5a;   
	 		Bandtype.Band_5b: r_goto_Fi := gc_r_band_5b ;
							  FeedIndexer.Status.p_Set:= gc_r_band_5b;   
	 		Bandtype.Band_6:  r_goto_Fi :=gc_r_band_6;
							  FeedIndexer.Status.p_Set:= gc_r_band_6;
;   
		END_CASE
	
		IF Move2Band = CmdResponseType.CommandActivated THEN  
			b_activate_Fi:=1;
			b_deactivate_Fi:=0;
			r_goto_v_Fi:= r_vel_max_Fi; 
			b_stop_Fi:= FALSE;
			b_start_goto_Fi:= TRUE;
			b_Move2Band_deactivate:= TRUE;
			Move2Band:=CmdResponseType.CommandActivated;
		ELSE 
			Move2Band:=CmdResponseType.ParameterOutOfRange;
		END_IF             			
							
	ELSE
		Move2Band:=CmdResponseType.CommandRejected;
		Command_Arbiter_error:=1;
	END_IF
END_IF

						

CommandArbiter.Status.LastCmdResponse:=Move2Band;
END_METHOD

METHOD Reset : UINT
VAR_INPUT
	SessionID: UINT;
	Axis: UINT;
END_VAR

VAR
	
END_VAR
CASE CommandArbiter.Status.DscCmdAuthority OF                    // Check that corerct user is issueing a command
	LMC: IF SessionID= CommandArbiter.Lmc_ID THEN
			Reset:= CmdResponseType.CommandActivated;
     	 END_IF
			
	EGUI: IF SessionID= CommandArbiter.Egui_ID THEN
			Reset:= CmdResponseType.CommandActivated;
    	  END_IF		
ELSE 
     Reset:= CmdResponseType.NoCmdAuth;
     Command_Arbiter_error:=1;	
END_CASE

IF Reset = CmdResponseType.CommandActivated THEN
	Command_Arbiter_error:=0;
	CASE Management.Status.DscState OF 
		DSCStateType.StartUp:
		 	Reset := CmdResponseType.CommandActivated;
		DSCStateType.Standby:
		 	Reset := CmdResponseType.CommandActivated;
		DSCStateType.Locked:
		 	Reset := CmdResponseType.CommandActivated;
		DSCStateType.Stowed:
		 	Reset :=CmdResponseType.CommandActivated;
		DSCStateType.Locked_Stowed:
		 	Reset := CmdResponseType.CommandActivated;
		DSCStateType.Activating :
		 	Reset := CmdResponseType.CommandRejected;
		DSCStateType.Deactivating :
		 	Reset := CmdResponseType.CommandRejected;
		DSCStateType.Standstill :
		 	Reset := CmdResponseType.CommandRejected;
		DSCStateType.Stopping :
		 	Reset := CmdResponseType.CommandRejected;
		DSCStateType.Slew :
		 	Reset := CmdResponseType.CommandRejected;
		DSCStateType.Jog :
		 	Reset := CmdResponseType.CommandRejected;
		DSCStateType.Track :
		 	Reset := CmdResponseType.CommandRejected;
	END_CASE

	IF Reset = CmdResponseType.CommandActivated THEN
		CASE Axis OF
			AxisSelectType.Az: b_clear_err_Az:= 1;
			AxisSelectType.El: b_clear_err_El:= 1;
			AxisSelectType.Fi: b_clear_err_Fi:= 1;
			AxisSelectType.AzEl: b_clear_err_Az:= 1;
								 b_clear_err_El:= 1;
			AxisSelectType.Unknown: b_clear_err:= 1;
		ELSE
			Reset := CmdResponseType.ParameterOutOfRange;
		END_CASE
	END_IF 
ELSE 
	 Reset:= CmdResponseType.NoCmdAuth;

END_IF

CommandArbiter.Status.LastCmdResponse:=Reset;
END_METHOD

METHOD SetOnSourceThreshold : Uint
VAR_INPUT
	SessionID :UINT;
	OnSourceThreshold : LREAL;
    ThresholdTimePeriod : LREAL;
END_VAR
CASE CommandArbiter.Status.DscCmdAuthority OF                    // Check that corerct user is issueing a command
	LMC: IF SessionID= CommandArbiter.Lmc_ID THEN
			SetOnSourceThreshold:= CmdResponseType.CommandActivated;
     	 END_IF
			
	EGUI: IF SessionID= CommandArbiter.Egui_ID THEN
			SetOnSourceThreshold:= CmdResponseType.CommandActivated;
    	  END_IF		
ELSE 
     SetOnSourceThreshold:= CmdResponseType.NoCmdAuth;
     Command_Arbiter_error:=1;	
END_CASE

IF SetOnSourceThreshold = CmdResponseType.CommandActivated THEN
	IF (OnSourceThreshold > 0 AND Onsourcethreshold <=20) OR ( ThresholdTimePeriod > 0 AND ThresholdTimePeriod <=10) THEN
		Tracking.Status.OnSourceThreshold:= OnSourceThreshold;
		Tracking.Status.ThresholdTimePeriod:=ThresholdTimePeriod;
		 t_onsource_dev_filt:=LREAL_TO_TIME(ThresholdTimePeriod*1000);
	    command_Arbiter_error:=0;
	ELSE
		SetOnSourceThreshold:= CmdResponseType.ParameterOutOfRange;
		Command_Arbiter_error:=1;
	END_IF
	
ELSE 
	 SetOnSourceThreshold:= CmdResponseType.CommandFailed;
	  Command_Arbiter_error:=1;
END_IF

CommandArbiter.Status.LastCmdResponse:=SetOnSourceThreshold;
END_METHOD

METHOD SetPowerMode : UINT (* Command to set the power mode *)
VAR_INPUT
	SessionID: UINT; (*Seesion ID*)
    LowPowerOn: BOOL:= FALSE; (* True = Low Power mode On *)
    PowerLimKw: LREAL:=10; (* Maximum Power limit in High power Mode *)

END_VAR
CASE CommandArbiter.Status.DscCmdAuthority OF                    // Check that correct user is issueing a command
	LMC: IF SessionID= CommandArbiter.Lmc_ID THEN
			SetPowerMode:= CmdResponseType.CommandActivated;
     	 END_IF
			
	EGUI: IF SessionID= CommandArbiter.Egui_ID THEN
			SetPowerMode:= CmdResponseType.CommandActivated;
    	  END_IF		
ELSE 
     SetPowerMode:= CmdResponseType.NoCmdAuth;
     Command_Arbiter_error:=1;	
END_CASE

IF SetPowerMode = CmdResponseType.CommandActivated THEN       // Check Dish State
	Command_Arbiter_error:=0;
	CASE Management.Status.DscState OF 
		DSCStateType.StartUp:
		 	SetPowerMode := CmdResponseType.CommandRejected;
		DSCStateType.Standby:
		 	SetPowerMode := CmdResponseType.CommandActivated;
		DSCStateType.Locked:
		 	SetPowerMode := CmdResponseType.CommandActivated;
		DSCStateType.Stowed:
		 	SetPowerMode :=CmdResponseType.CommandActivated;
		DSCStateType.Locked_Stowed:
		 	SetPowerMode := CmdResponseType.CommandActivated;
		DSCStateType.Activating :
		 	SetPowerMode := CmdResponseType.CommandActivated;
		DSCStateType.Deactivating :
		 	SetPowerMode := CmdResponseType.CommandActivated;
		DSCStateType.Standstill :
		 	SetPowerMode := CmdResponseType.CommandActivated;
		DSCStateType.Stopping :
		 	SetPowerMode := CmdResponseType.CommandActivated;
		DSCStateType.Slew :
		 	SetPowerMode := CmdResponseType.CommandActivated;
		DSCStateType.Jog :
		 	SetPowerMode := CmdResponseType.CommandActivated;
		DSCStateType.Track :
		 	SetPowerMode := CmdResponseType.CommandActivated;
	END_CASE
END_IF

IF SetPowerMode = CmdResponseType.CommandActivated THEN
	//SetPowerMode := CmdResponseType.NotImplemented;
	IF LowPowerOn =1 THEN 
		Management.PowerStatus.LowPowerActive:=1;
		IF Azimuth.Status.Active THEN
			b_deactivate_Az:=1;
			b_activate_Az:=0;
		END_IF
		
		IF Elevation.Status.Active THEN
			b_deactivate_El:=1;
			b_activate_El:=0;
		END_IF
		
		IF FeedIndexer.Status.Active THEN
			b_deactivate_Fi:=1;
	    	b_activate_Fi:=0;
		END_IF 
					
	ELSE
		Management.PowerStatus.LowPowerActive:=0;
		r_vel_max_Az:=  gc_r_power_Kv_Az*PowerLimKw;
  		r_vel_max_El:=  gc_r_power_Kv_El*PowerLimKw;
  		r_vel_max_Fi:=  gc_r_power_Kv_Fi*PowerLimKw;
		r_goto_acc_Az:= gc_r_power_Ka_Az*PowerLimKw;
  		r_goto_acc_El:= gc_r_power_Ka_El*PowerLimKw;
  		r_goto_acc_Fi:= gc_r_power_Ka_Fi*PowerLimKw;
  	END_IF
END_IF

CommandArbiter.Status.LastCmdResponse:=SetPowerMode;
END_METHOD

METHOD Slew2AbsSingleAx : UINT
VAR_INPUT
	SessionID: UINT;
	Axis: Uint;
	Position:LREAL;
	Speed:LREAL;
END_VAR

VAR
END_VAR
CASE CommandArbiter.Status.DscCmdAuthority OF                    // Check that correct user is issueing a command
	LMC: IF SessionID= CommandArbiter.Lmc_ID THEN
			Slew2AbsSingleAx:= CmdResponseType.CommandActivated;
     	 END_IF
			
	EGUI: IF SessionID= CommandArbiter.Egui_ID THEN
			Slew2AbsSingleAx:= CmdResponseType.CommandActivated;
    	  END_IF		
ELSE 
     Slew2AbsSingleAx:= CmdResponseType.NoCmdAuth;
     Command_Arbiter_error:=1;	
END_CASE

IF Slew2AbsSingleAx = CmdResponseType.CommandActivated THEN // Dish State to see if move is possible
	Command_Arbiter_error:=0;
	//IF  Management.ErrorStatus.errGeneral=0 AND Management.WarningStatus.waMngmnt =0 THEN   If the Dish has errors that prevent movement then it will not be in a state where it can be moved. 
		CASE Management.Status.DscState OF 
			 DscStateType.Locked:        Slew2AbsSingleAx:=CmdResponseType.DishLocked;
			 DscStateType.Locked_Stowed: Slew2AbsSingleAx:=CmdResponseType.DishLocked;
			 DscStateType.Standstill:    Slew2AbsSingleAx:=CmdResponseType.CommandActivated;
		     DscStateType.Standby:       Slew2AbsSingleAx:=CmdResponseType.CommandActivated;
			 DscStateType.Stowed:	IF Axis=2 THEN 
				Slew2AbsSingleAx:= CmdResponseType.CommandActivated;
			ELSE
		 	Slew2AbsSingleAx:=CmdResponseType.Stowed;
			END_IF
  
		ELSE
		     Slew2AbsSingleAx:=CmdResponseType.CommandRejected;
		     Command_Arbiter_error:=1;
		END_CASE								
	//ELSE
	//	Slew2AbsAx:=CmdResponseType.CommandAborted;
	//	Command_Arbiter_error:=1;
	//END_IF
END_IF
	
